	SBR_A_4_FowardDecant_XV26 AT%Q* : BOOL;
	SBR_A_4_ReverseDecant_XV26 AT%Q* : BOOL;
	SBR_A_4_BlowerValve_XV201 AT%Q* : BOOL;
	SBR_A_4_DeSludgeValve_XV241 AT%Q* : BOOL;
	SBR_A_4_SBRValve_XV205 AT%Q* : BOOL;
	SBR_A_4_SBRMixer_XV205 : BOOL;

	SBR_A_4_bEnable_SW : BOOL;
	SBR_A_4_Blower_B201 : BOOL;
	SBR_A_4_DesludgePump_P201 : BOOL;
	SBR_A_4_filling : BOOL;
	SBR_A_4_aeration : BOOL;
	SBR_A_4_settling : BOOL;
	SBR_A_4_decanting : BOOL;
	SBR_A_4_desludging : BOOL;
	SBR_A_4_SBRMixer_M200 : BOOL;
	SBR_A_4_warning_DONotInRange : BOOL;


	SludeTankSensorLevelHi_LSL510A: inBlock;
	SBRReactor_1: SBRReactor;
	SBRReactor_2: SBRReactor;
	SBRReactor_3: SBRReactor;
	SBRReactor_4: SBRReactor;

	SBRMixer_M200A1_A_remote_mode AT%I* : BOOL;
	SBRMixer_M200A1_A_overload AT%I* : BOOL;
	SBRMixer_M200A1_A_incomplete AT%I* : BOOL;
	SBRMixer_M200A1_A_status AT%I* : BOOL;

	SBRMixer_M200A1_A_command AT%Q* : BOOL;

	SBRMixer_M200A1_A_in : BOOL;
	SBRMixer_M200A1_A_overload_error : BOOL;
	SBRMixer_M200A1_A_incomplete_error : BOOL;
	SBRMixer_M200A1_A_status_error : BOOL;
	SBRMixer_M200A1_A_common_error : BOOL;
	SBRMixer_M200A1_A_stop_error : BOOL;

	SBRMixer_M200A1_A_overload_Filter : ErrorFilter;
	SBRMixer_M200A1_A_incomplete_Filter : ErrorFilter;
	SBRMixer_M200A1_A_status_Filter : ErrorFilter;
	SBRMixer_M200A1_A_stop_Filter : ErrorFilter;

	SBRMixer_M200A1_B_remote_mode AT%I* : BOOL;
	SBRMixer_M200A1_B_overload AT%I* : BOOL;
	SBRMixer_M200A1_B_incomplete AT%I* : BOOL;
	SBRMixer_M200A1_B_status AT%I* : BOOL;

	SBRMixer_M200A1_B_command AT%Q* : BOOL;

	SBRMixer_M200A1_B_in : BOOL;
	SBRMixer_M200A1_B_overload_error : BOOL;
	SBRMixer_M200A1_B_incomplete_error : BOOL;
	SBRMixer_M200A1_B_status_error : BOOL;
	SBRMixer_M200A1_B_common_error : BOOL;
	SBRMixer_M200A1_B_stop_error : BOOL;

	SBRMixer_M200A1_B_overload_Filter : ErrorFilter;
	SBRMixer_M200A1_B_incomplete_Filter : ErrorFilter;
	SBRMixer_M200A1_B_status_Filter : ErrorFilter;
	SBRMixer_M200A1_B_stop_Filter : ErrorFilter;


	SBRMixer_M200A1_C_remote_mode AT%I* : BOOL;
	SBRMixer_M200A1_C_overload AT%I* : BOOL;
	SBRMixer_M200A1_C_incomplete AT%I* : BOOL;
	SBRMixer_M200A1_C_status AT%I* : BOOL;

	SBRMixer_M200A1_C_command AT%Q* : BOOL;

	SBRMixer_M200A1_C_in : BOOL;
	SBRMixer_M200A1_C_overload_error : BOOL;
	SBRMixer_M200A1_C_incomplete_error : BOOL;
	SBRMixer_M200A1_C_status_error : BOOL;
	SBRMixer_M200A1_C_common_error : BOOL;
	SBRMixer_M200A1_C_stop_error : BOOL;

	SBRMixer_M200A1_C_overload_Filter : ErrorFilter;
	SBRMixer_M200A1_C_incomplete_Filter : ErrorFilter;
	SBRMixer_M200A1_C_status_Filter : ErrorFilter;
	SBRMixer_M200A1_C_stop_Filter : ErrorFilter;



	SBRMixer_M200A2_A_remote_mode AT%I* : BOOL;
	SBRMixer_M200A2_A_overload AT%I* : BOOL;
	SBRMixer_M200A2_A_incomplete AT%I* : BOOL;
	SBRMixer_M200A2_A_status AT%I* : BOOL;

	SBRMixer_M200A2_A_command AT%Q* : BOOL;

	SBRMixer_M200A2_A_in : BOOL;
	SBRMixer_M200A2_A_overload_error : BOOL;
	SBRMixer_M200A2_A_incomplete_error : BOOL;
	SBRMixer_M200A2_A_status_error : BOOL;
	SBRMixer_M200A2_A_common_error : BOOL;
	SBRMixer_M200A2_A_stop_error : BOOL;

	SBRMixer_M200A2_A_overload_Filter : ErrorFilter;
	SBRMixer_M200A2_A_incomplete_Filter : ErrorFilter;
	SBRMixer_M200A2_A_status_Filter : ErrorFilter;
	SBRMixer_M200A2_A_stop_Filter : ErrorFilter;

	SBRMixer_M200A2_B_remote_mode AT%I* : BOOL;
	SBRMixer_M200A2_B_overload AT%I* : BOOL;
	SBRMixer_M200A2_B_incomplete AT%I* : BOOL;
	SBRMixer_M200A2_B_status AT%I* : BOOL;

	SBRMixer_M200A2_B_command AT%Q* : BOOL;

	SBRMixer_M200A2_B_in : BOOL;
	SBRMixer_M200A2_B_overload_error : BOOL;
	SBRMixer_M200A2_B_incomplete_error : BOOL;
	SBRMixer_M200A2_B_status_error : BOOL;
	SBRMixer_M200A2_B_common_error : BOOL;
	SBRMixer_M200A2_B_stop_error : BOOL;

	SBRMixer_M200A2_B_overload_Filter : ErrorFilter;
	SBRMixer_M200A2_B_incomplete_Filter : ErrorFilter;
	SBRMixer_M200A2_B_status_Filter : ErrorFilter;
	SBRMixer_M200A2_B_stop_Filter : ErrorFilter;


	SBRMixer_M200A2_C_remote_mode AT%I* : BOOL;
	SBRMixer_M200A2_C_overload AT%I* : BOOL;
	SBRMixer_M200A2_C_incomplete AT%I* : BOOL;
	SBRMixer_M200A2_C_status AT%I* : BOOL;

	SBRMixer_M200A2_C_command AT%Q* : BOOL;

	SBRMixer_M200A2_C_in : BOOL;
	SBRMixer_M200A2_C_overload_error : BOOL;
	SBRMixer_M200A2_C_incomplete_error : BOOL;
	SBRMixer_M200A2_C_status_error : BOOL;
	SBRMixer_M200A2_C_common_error : BOOL;
	SBRMixer_M200A2_C_stop_error : BOOL;

	SBRMixer_M200A2_C_overload_Filter : ErrorFilter;
	SBRMixer_M200A2_C_incomplete_Filter : ErrorFilter;
	SBRMixer_M200A2_C_status_Filter : ErrorFilter;
	SBRMixer_M200A2_C_stop_Filter : ErrorFilter;



	SBRMixer_M200A3_A_remote_mode AT%I* : BOOL;
	SBRMixer_M200A3_A_overload AT%I* : BOOL;
	SBRMixer_M200A3_A_incomplete AT%I* : BOOL;
	SBRMixer_M200A3_A_status AT%I* : BOOL;

	SBRMixer_M200A3_A_command AT%Q* : BOOL;

	SBRMixer_M200A3_A_in : BOOL;
	SBRMixer_M200A3_A_overload_error : BOOL;
	SBRMixer_M200A3_A_incomplete_error : BOOL;
	SBRMixer_M200A3_A_status_error : BOOL;
	SBRMixer_M200A3_A_common_error : BOOL;
	SBRMixer_M200A3_A_stop_error : BOOL;

	SBRMixer_M200A3_A_overload_Filter : ErrorFilter;
	SBRMixer_M200A3_A_incomplete_Filter : ErrorFilter;
	SBRMixer_M200A3_A_status_Filter : ErrorFilter;
	SBRMixer_M200A3_A_stop_Filter : ErrorFilter;

	SBRMixer_M200A3_B_remote_mode AT%I* : BOOL;
	SBRMixer_M200A3_B_overload AT%I* : BOOL;
	SBRMixer_M200A3_B_incomplete AT%I* : BOOL;
	SBRMixer_M200A3_B_status AT%I* : BOOL;

	SBRMixer_M200A3_B_command AT%Q* : BOOL;

	SBRMixer_M200A3_B_in : BOOL;
	SBRMixer_M200A3_B_overload_error : BOOL;
	SBRMixer_M200A3_B_incomplete_error : BOOL;
	SBRMixer_M200A3_B_status_error : BOOL;
	SBRMixer_M200A3_B_common_error : BOOL;
	SBRMixer_M200A3_B_stop_error : BOOL;

	SBRMixer_M200A3_B_overload_Filter : ErrorFilter;
	SBRMixer_M200A3_B_incomplete_Filter : ErrorFilter;
	SBRMixer_M200A3_B_status_Filter : ErrorFilter;
	SBRMixer_M200A3_B_stop_Filter : ErrorFilter;


	SBRMixer_M200A3_C_remote_mode AT%I* : BOOL;
	SBRMixer_M200A3_C_overload AT%I* : BOOL;
	SBRMixer_M200A3_C_incomplete AT%I* : BOOL;
	SBRMixer_M200A3_C_status AT%I* : BOOL;

	SBRMixer_M200A3_C_command AT%Q* : BOOL;

	SBRMixer_M200A3_C_in : BOOL;
	SBRMixer_M200A3_C_overload_error : BOOL;
	SBRMixer_M200A3_C_incomplete_error : BOOL;
	SBRMixer_M200A3_C_status_error : BOOL;
	SBRMixer_M200A3_C_common_error : BOOL;
	SBRMixer_M200A3_C_stop_error : BOOL;

	SBRMixer_M200A3_C_overload_Filter : ErrorFilter;
	SBRMixer_M200A3_C_incomplete_Filter : ErrorFilter;
	SBRMixer_M200A3_C_status_Filter : ErrorFilter;
	SBRMixer_M200A3_C_stop_Filter : ErrorFilter;

	DesludgePump_P201A_1_remote_mode AT%I* : BOOL;
	DesludgePump_P201A_1_overload AT%I* : BOOL;
	DesludgePump_P201A_1_incomplete AT%I* : BOOL;
	DesludgePump_P201A_1_status AT%I* : BOOL;

	DesludgePump_P201A_1_command AT%Q* : BOOL;

	DesludgePump_P201A_1_in : BOOL;
	DesludgePump_P201A_1_overload_error : BOOL;
	DesludgePump_P201A_1_incomplete_error : BOOL;
	DesludgePump_P201A_1_status_error : BOOL;
	DesludgePump_P201A_1_common_error : BOOL;
	DesludgePump_P201A_1_stop_error : BOOL;

	DesludgePump_P201A_1_overload_Filter : ErrorFilter;
	DesludgePump_P201A_1_incomplete_Filter : ErrorFilter;
	DesludgePump_P201A_1_status_Filter : ErrorFilter;
	DesludgePump_P201A_1_stop_Filter : ErrorFilter;



	DesludgePump_P201A_2_remote_mode AT%I* : BOOL;
	DesludgePump_P201A_2_overload AT%I* : BOOL;
	DesludgePump_P201A_2_incomplete AT%I* : BOOL;
	DesludgePump_P201A_2_status AT%I* : BOOL;

	DesludgePump_P201A_2_command AT%Q* : BOOL;

	DesludgePump_P201A_2_in : BOOL;
	DesludgePump_P201A_2_overload_error : BOOL;
	DesludgePump_P201A_2_incomplete_error : BOOL;
	DesludgePump_P201A_2_status_error : BOOL;
	DesludgePump_P201A_2_common_error : BOOL;
	DesludgePump_P201A_2_stop_error : BOOL;

	DesludgePump_P201A_2_overload_Filter : ErrorFilter;
	DesludgePump_P201A_2_incomplete_Filter : ErrorFilter;
	DesludgePump_P201A_2_status_Filter : ErrorFilter;
	DesludgePump_P201A_2_stop_Filter : ErrorFilter;

	DesludgePump_P201A :Equipment_Dual;


	Blower_B201A_1_remote_mode AT%I* : BOOL;
	Blower_B201A_1_overload AT%I* : BOOL;
	Blower_B201A_1_incomplete AT%I* : BOOL;
	Blower_B201A_1_status AT%I* : BOOL;

	Blower_B201A_1_command AT%Q* : BOOL;

	Blower_B201A_1_in : BOOL;
	Blower_B201A_1_overload_error : BOOL;
	Blower_B201A_1_incomplete_error : BOOL;
	Blower_B201A_1_status_error : BOOL;
	Blower_B201A_1_common_error : BOOL;
	Blower_B201A_1_stop_error : BOOL;

	Blower_B201A_1_overload_Filter : ErrorFilter;
	Blower_B201A_1_incomplete_Filter : ErrorFilter;
	Blower_B201A_1_status_Filter : ErrorFilter;
	Blower_B201A_1_stop_Filter : ErrorFilter;



	Blower_B201A_2_remote_mode AT%I* : BOOL;
	Blower_B201A_2_overload AT%I* : BOOL;
	Blower_B201A_2_incomplete AT%I* : BOOL;
	Blower_B201A_2_status AT%I* : BOOL;

	Blower_B201A_2_command AT%Q* : BOOL;

	Blower_B201A_2_in : BOOL;
	Blower_B201A_2_overload_error : BOOL;
	Blower_B201A_2_incomplete_error : BOOL;
	Blower_B201A_2_status_error : BOOL;
	Blower_B201A_2_common_error : BOOL;
	Blower_B201A_2_stop_error : BOOL;

	Blower_B201A_2_overload_Filter : ErrorFilter;
	Blower_B201A_2_incomplete_Filter : ErrorFilter;
	Blower_B201A_2_status_Filter : ErrorFilter;
	Blower_B201A_2_stop_Filter : ErrorFilter;



	Blower_B201A_3_remote_mode AT%I* : BOOL;
	Blower_B201A_3_overload AT%I* : BOOL;
	Blower_B201A_3_incomplete AT%I* : BOOL;
	Blower_B201A_3_status AT%I* : BOOL;

	Blower_B201A_3_command AT%Q* : BOOL;

	Blower_B201A_3_in : BOOL;
	Blower_B201A_3_overload_error : BOOL;
	Blower_B201A_3_incomplete_error : BOOL;
	Blower_B201A_3_status_error : BOOL;
	Blower_B201A_3_common_error : BOOL;
	Blower_B201A_3_stop_error : BOOL;

	Blower_B201A_3_overload_Filter : ErrorFilter;
	Blower_B201A_3_incomplete_Filter : ErrorFilter;
	Blower_B201A_3_status_Filter : ErrorFilter;
	Blower_B201A_3_stop_Filter : ErrorFilter;


END_VAR

VAR PERSISTENT
	FILLING_TOKEN : INT;
	AERATION_TOKEN: INT;
	DECANTING_TOKEN: INT;
END_VAR
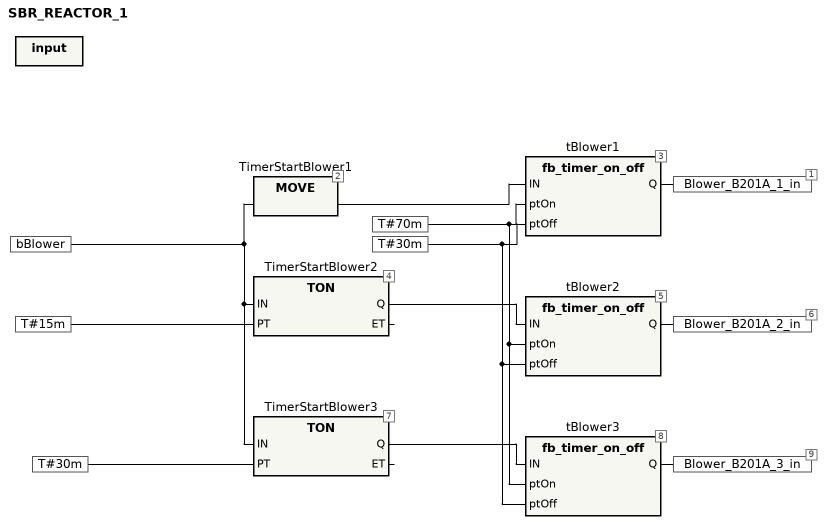
[picture p10: SBR_REACTOR_1 (CFC)]
_CFC_ (* Continuous Function Chart, elements in execution order *)
#0 input()
#1 Blower_B201A_1_in <= #3.Q
#2 TimerStartBlower1:MOVE(bBlower)
#3 tBlower1:fb_timer_on_off(IN: #2, ptOn: T#70m, ptOff: T#30m)
#4 TimerStartBlower2:TON(IN: bBlower, PT: T#15m)
#5 tBlower2:fb_timer_on_off(IN: #4.Q, ptOn: T#70m, ptOff: T#30m)
#6 Blower_B201A_2_in <= #5.Q
#7 TimerStartBlower3:TON(IN: bBlower, PT: T#30m)
#8 tBlower3:fb_timer_on_off(IN: #7.Q, ptOn: T#70m, ptOff: T#30m)
#9 Blower_B201A_3_in <= #8.Q
_END_CFC_
END_PROGRAM
ACTION input:
SludeTankSensorLevelHi_LSL510A();

SBRReactor_1(
	bEnable:=SBR_A_1_bEnable_SW ,
	SludgeTankLevelHi:= SludeTankSensorLevelHi_LSL510A.Q,
	SBRLevelSensor_LSH200:= SBR_A_1_SBRLevelSensor_LSH200,
	rDO201:= SBR_A_1_DOSensor_DO201,
	DecanterLevelSensorHi:=SBR_A_1_DecanterLevelSensorHi_Rx ,
	DecanterLevelSensorLow:=SBR_A_1_DecanterLevelSensorLow_Rx ,
	FILLING_TOKEN:=FILLING_TOKEN ,
	AERATION_TOKEN:= AERATION_TOKEN,
	DECANTING_TOKEN:= DECANTING_TOKEN,
	bBlowerOn=>SBR_A_1_Blower_B201 ,
	bDeSludgePump=>SBR_A_1_DesludgePump_P201 ,
	bFilling=>SBR_A_1_filling ,
	bAeration=>SBR_A_1_aeration ,
	bSettling=>SBR_A_1_settling ,
	bDecanting=>SBR_A_1_decanting ,
	bDesluging=>SBR_A_1_desludging ,
	bWarning_DoNotInRange=>SBR_A_1_warning_DONotInRange ,
	bForwardDecant=>SBR_A_1_FowardDecant_XV26 ,
	bReverseDecant=>SBR_A_1_ReverseDecant_XV26 ,
	bBlowerValve_XV201=>SBR_A_1_BlowerValve_XV201 ,
	bDeslugValve_XV241=> SBR_A_1_DeSludgeValve_XV241,
	bSBRValve_XV205=>SBR_A_1_SBRValve_XV205 ,
	bSBRMixer=>SBR_A_1_SBRMixer_XV205 );


SBRReactor_2(
	bEnable:=SBR_A_2_bEnable_SW ,
	SludgeTankLevelHi:= SludeTankSensorLevelHi_LSL510A.Q,
	SBRLevelSensor_LSH200:= SBR_A_2_SBRLevelSensor_LSH200,
	rDO201:= SBR_A_2_DOSensor_DO201,
	DecanterLevelSensorHi:=SBR_A_2_DecanterLevelSensorHi_Rx ,
	DecanterLevelSensorLow:=SBR_A_2_DecanterLevelSensorLow_Rx ,
	FILLING_TOKEN:=FILLING_TOKEN ,
	AERATION_TOKEN:= AERATION_TOKEN,
	DECANTING_TOKEN:= DECANTING_TOKEN,
	bBlowerOn=>SBR_A_2_Blower_B201 ,
	bDeSludgePump=>SBR_A_2_DesludgePump_P201 ,
	bFilling=>SBR_A_2_filling ,
	bAeration=>SBR_A_2_aeration ,
	bSettling=>SBR_A_2_settling ,
	bDecanting=>SBR_A_2_decanting ,
	bDesluging=>SBR_A_2_desludging ,
	bWarning_DoNotInRange=>SBR_A_2_warning_DONotInRange ,
	bForwardDecant=>SBR_A_2_FowardDecant_XV26 ,
	bReverseDecant=>SBR_A_2_ReverseDecant_XV26 ,
	bBlowerValve_XV201=>SBR_A_2_BlowerValve_XV201 ,
	bDeslugValve_XV241=> SBR_A_2_DeSludgeValve_XV241,
	bSBRValve_XV205=>SBR_A_2_SBRValve_XV205 ,
	bSBRMixer=>SBR_A_2_SBRMixer_XV205 );


SBRReactor_3(
	bEnable:=SBR_A_3_bEnable_SW ,
	SludgeTankLevelHi:= SludeTankSensorLevelHi_LSL510A.Q,
	SBRLevelSensor_LSH200:= SBR_A_3_SBRLevelSensor_LSH200,
	rDO201:= SBR_A_3_DOSensor_DO201,
	DecanterLevelSensorHi:=SBR_A_3_DecanterLevelSensorHi_Rx ,
	DecanterLevelSensorLow:=SBR_A_3_DecanterLevelSensorLow_Rx ,
	FILLING_TOKEN:=FILLING_TOKEN ,
	AERATION_TOKEN:= AERATION_TOKEN,
	DECANTING_TOKEN:= DECANTING_TOKEN,
	bBlowerOn=>SBR_A_3_Blower_B201 ,
	bDeSludgePump=>SBR_A_3_DesludgePump_P201 ,
	bFilling=>SBR_A_3_filling ,
	bAeration=>SBR_A_3_aeration ,
	bSettling=>SBR_A_3_settling ,
	bDecanting=>SBR_A_3_decanting ,
	bDesluging=>SBR_A_3_desludging ,
	bWarning_DoNotInRange=>SBR_A_3_warning_DONotInRange ,
	bForwardDecant=>SBR_A_3_FowardDecant_XV26 ,
	bReverseDecant=>SBR_A_3_ReverseDecant_XV26 ,
	bBlowerValve_XV201=>SBR_A_3_BlowerValve_XV201 ,
	bDeslugValve_XV241=> SBR_A_3_DeSludgeValve_XV241,
	bSBRValve_XV205=>SBR_A_3_SBRValve_XV205 ,
	bSBRMixer=>SBR_A_3_SBRMixer_XV205 );


SBRReactor_4(
	bEnable:=SBR_A_4_bEnable_SW ,
	SludgeTankLevelHi:= SludeTankSensorLevelHi_LSL510A.Q,
	SBRLevelSensor_LSH200:= SBR_A_4_SBRLevelSensor_LSH200,
	rDO201:= SBR_A_4_DOSensor_DO201,
	DecanterLevelSensorHi:=SBR_A_4_DecanterLevelSensorHi_Rx ,
	DecanterLevelSensorLow:=SBR_A_4_DecanterLevelSensorLow_Rx ,
	FILLING_TOKEN:=FILLING_TOKEN ,
	AERATION_TOKEN:= AERATION_TOKEN,
	DECANTING_TOKEN:= DECANTING_TOKEN,
	bBlowerOn=>SBR_A_4_Blower_B201 ,
	bDeSludgePump=>SBR_A_4_DesludgePump_P201 ,
	bFilling=>SBR_A_4_filling ,
	bAeration=>SBR_A_4_aeration ,
	bSettling=>SBR_A_4_settling ,
	bDecanting=>SBR_A_4_decanting ,
	bDesluging=>SBR_A_4_desludging ,
	bWarning_DoNotInRange=>SBR_A_4_warning_DONotInRange ,
	bForwardDecant=>SBR_A_4_FowardDecant_XV26 ,
	bReverseDecant=>SBR_A_4_ReverseDecant_XV26 ,
	bBlowerValve_XV201=>SBR_A_4_BlowerValve_XV201 ,
	bDeslugValve_XV241=> SBR_A_4_DeSludgeValve_XV241,
	bSBRValve_XV205=>SBR_A_4_SBRValve_XV205 ,
	bSBRMixer=>SBR_A_4_SBRMixer_XV205 );


bDeSludge:=SBR_A_1_DeSludgeValve_XV241 OR SBR_A_2_DeSludgeValve_XV241 OR SBR_A_3_DeSludgeValve_XV241 OR SBR_A_4_DeSludgeValve_XV241;
bBlower:= SBR_A_1_Blower_B201 OR SBR_A_2_Blower_B201 OR SBR_A_3_Blower_B201 OR SBR_A_4_Blower_B201;



SBRMixer_M200A1_A_in := SBR_A_1_SBRMixer_XV205;
SBRMixer_M200A1_A_command := SBRMixer_M200A1_A_in AND SBRMixer_M200A1_A_remote_mode;
SBRMixer_M200A1_A_overload_Filter(IN:=(SBRMixer_M200A1_A_overload AND SBRMixer_M200A1_A_in),PT:=T#2s,Q=>SBRMixer_M200A1_A_overload_error);
SBRMixer_M200A1_A_incomplete_Filter(IN:=(SBRMixer_M200A1_A_incomplete AND SBRMixer_M200A1_A_in),PT:=T#2s,Q=>SBRMixer_M200A1_A_incomplete_error);
SBRMixer_M200A1_A_status_Filter(IN:=(NOT SBRMixer_M200A1_A_status AND SBRMixer_M200A1_A_in),PT:=T#10s, Q=>SBRMixer_M200A1_A_status_error);
SBRMixer_M200A1_A_stop_Filter(IN:=( SBRMixer_M200A1_A_status AND NOT SBRMixer_M200A1_A_in),PT:=T#10s, Q=>SBRMixer_M200A1_A_stop_error);

SBRMixer_M200A1_A_common_error := SBRMixer_M200A1_A_overload_error OR SBRMixer_M200A1_A_incomplete_error OR SBRMixer_M200A1_A_status_error OR SBRMixer_M200A1_A_stop_error;


SBRMixer_M200A1_B_in := SBR_A_1_SBRMixer_XV205;
SBRMixer_M200A1_B_command := SBRMixer_M200A1_B_in AND SBRMixer_M200A1_B_remote_mode;
SBRMixer_M200A1_B_overload_Filter(IN:=(SBRMixer_M200A1_B_overload AND SBRMixer_M200A1_B_in),PT:=T#2s,Q=>SBRMixer_M200A1_B_overload_error);
SBRMixer_M200A1_B_incomplete_Filter(IN:=(SBRMixer_M200A1_B_incomplete AND SBRMixer_M200A1_B_in),PT:=T#2s,Q=>SBRMixer_M200A1_B_incomplete_error);
SBRMixer_M200A1_B_status_Filter(IN:=(NOT SBRMixer_M200A1_B_status AND SBRMixer_M200A1_B_in),PT:=T#10s, Q=>SBRMixer_M200A1_B_status_error);
SBRMixer_M200A1_B_stop_Filter(IN:=( SBRMixer_M200A1_B_status AND NOT SBRMixer_M200A1_B_in),PT:=T#10s, Q=>SBRMixer_M200A1_B_stop_error);

SBRMixer_M200A1_B_common_error := SBRMixer_M200A1_B_overload_error OR SBRMixer_M200A1_B_incomplete_error OR SBRMixer_M200A1_B_status_error OR SBRMixer_M200A1_B_stop_error;


SBRMixer_M200A1_C_in := SBR_A_1_SBRMixer_XV205;
SBRMixer_M200A1_C_command := SBRMixer_M200A1_C_in AND SBRMixer_M200A1_C_remote_mode;
SBRMixer_M200A1_C_overload_Filter(IN:=(SBRMixer_M200A1_C_overload AND SBRMixer_M200A1_C_in),PT:=T#2s,Q=>SBRMixer_M200A1_C_overload_error);
SBRMixer_M200A1_C_incomplete_Filter(IN:=(SBRMixer_M200A1_C_incomplete AND SBRMixer_M200A1_C_in),PT:=T#2s,Q=>SBRMixer_M200A1_C_incomplete_error);
SBRMixer_M200A1_C_status_Filter(IN:=(NOT SBRMixer_M200A1_C_status AND SBRMixer_M200A1_C_in),PT:=T#10s, Q=>SBRMixer_M200A1_C_status_error);
SBRMixer_M200A1_C_stop_Filter(IN:=( SBRMixer_M200A1_C_status AND NOT SBRMixer_M200A1_C_in),PT:=T#10s, Q=>SBRMixer_M200A1_C_stop_error);

SBRMixer_M200A1_C_common_error := SBRMixer_M200A1_C_overload_error OR SBRMixer_M200A1_C_incomplete_error OR SBRMixer_M200A1_C_status_error OR SBRMixer_M200A1_C_stop_error;



SBRMixer_M200A2_A_in := SBR_A_2_SBRMixer_XV205;
SBRMixer_M200A2_A_command := SBRMixer_M200A2_A_in AND SBRMixer_M200A2_A_remote_mode;
SBRMixer_M200A2_A_overload_Filter(IN:=(SBRMixer_M200A2_A_overload AND SBRMixer_M200A2_A_in),PT:=T#2s,Q=>SBRMixer_M200A2_A_overload_error);
SBRMixer_M200A2_A_incomplete_Filter(IN:=(SBRMixer_M200A2_A_incomplete AND SBRMixer_M200A2_A_in),PT:=T#2s,Q=>SBRMixer_M200A2_A_incomplete_error);
SBRMixer_M200A2_A_status_Filter(IN:=(NOT SBRMixer_M200A2_A_status AND SBRMixer_M200A2_A_in),PT:=T#10s, Q=>SBRMixer_M200A2_A_status_error);
SBRMixer_M200A2_A_stop_Filter(IN:=( SBRMixer_M200A2_A_status AND NOT SBRMixer_M200A2_A_in),PT:=T#10s, Q=>SBRMixer_M200A2_A_stop_error);

SBRMixer_M200A2_A_common_error := SBRMixer_M200A2_A_overload_error OR SBRMixer_M200A2_A_incomplete_error OR SBRMixer_M200A2_A_status_error OR SBRMixer_M200A2_A_stop_error;


SBRMixer_M200A2_B_in := SBR_A_2_SBRMixer_XV205;
SBRMixer_M200A2_B_command := SBRMixer_M200A2_B_in AND SBRMixer_M200A2_B_remote_mode;
SBRMixer_M200A2_B_overload_Filter(IN:=(SBRMixer_M200A2_B_overload AND SBRMixer_M200A2_B_in),PT:=T#2s,Q=>SBRMixer_M200A2_B_overload_error);
SBRMixer_M200A2_B_incomplete_Filter(IN:=(SBRMixer_M200A2_B_incomplete AND SBRMixer_M200A2_B_in),PT:=T#2s,Q=>SBRMixer_M200A2_B_incomplete_error);
SBRMixer_M200A2_B_status_Filter(IN:=(NOT SBRMixer_M200A2_B_status AND SBRMixer_M200A2_B_in),PT:=T#10s, Q=>SBRMixer_M200A2_B_status_error);
SBRMixer_M200A1_B_stop_Filter(IN:=( SBRMixer_M200A1_B_status AND NOT SBRMixer_M200A1_B_in),PT:=T#10s, Q=>SBRMixer_M200A1_B_stop_error);

SBRMixer_M200A1_B_common_error := SBRMixer_M200A1_B_overload_error OR SBRMixer_M200A1_B_incomplete_error OR SBRMixer_M200A1_B_status_error OR SBRMixer_M200A1_B_stop_error;


SBRMixer_M200A2_C_in := SBR_A_2_SBRMixer_XV205;
SBRMixer_M200A2_C_command := SBRMixer_M200A2_C_in AND SBRMixer_M200A2_C_remote_mode;
SBRMixer_M200A2_C_overload_Filter(IN:=(SBRMixer_M200A2_C_overload AND SBRMixer_M200A2_C_in),PT:=T#2s,Q=>SBRMixer_M200A2_C_overload_error);
SBRMixer_M200A2_C_incomplete_Filter(IN:=(SBRMixer_M200A2_C_incomplete AND SBRMixer_M200A2_C_in),PT:=T#2s,Q=>SBRMixer_M200A2_C_incomplete_error);
SBRMixer_M200A2_C_status_Filter(IN:=(NOT SBRMixer_M200A2_C_status AND SBRMixer_M200A2_C_in),PT:=T#10s, Q=>SBRMixer_M200A2_C_status_error);
SBRMixer_M200A2_C_stop_Filter(IN:=( SBRMixer_M200A2_C_status AND NOT SBRMixer_M200A2_C_in),PT:=T#10s, Q=>SBRMixer_M200A2_C_stop_error);

SBRMixer_M200A2_C_common_error := SBRMixer_M200A2_C_overload_error OR SBRMixer_M200A2_C_incomplete_error OR SBRMixer_M200A2_C_status_error OR SBRMixer_M200A2_C_stop_error;



SBRMixer_M200A3_A_in := SBR_A_3_SBRMixer_XV205;
SBRMixer_M200A3_A_command := SBRMixer_M200A3_A_in AND SBRMixer_M200A3_A_remote_mode;
SBRMixer_M200A3_A_overload_Filter(IN:=(SBRMixer_M200A3_A_overload AND SBRMixer_M200A3_A_in),PT:=T#2s,Q=>SBRMixer_M200A3_A_overload_error);
SBRMixer_M200A3_A_incomplete_Filter(IN:=(SBRMixer_M200A3_A_incomplete AND SBRMixer_M200A3_A_in),PT:=T#2s,Q=>SBRMixer_M200A3_A_incomplete_error);
SBRMixer_M200A3_A_status_Filter(IN:=(NOT SBRMixer_M200A3_A_status AND SBRMixer_M200A3_A_in),PT:=T#10s, Q=>SBRMixer_M200A3_A_status_error);
SBRMixer_M200A3_A_stop_Filter(IN:=( SBRMixer_M200A3_A_status AND NOT SBRMixer_M200A3_A_in),PT:=T#10s, Q=>SBRMixer_M200A3_A_stop_error);

SBRMixer_M200A3_A_common_error := SBRMixer_M200A3_A_overload_error OR SBRMixer_M200A3_A_incomplete_error OR SBRMixer_M200A3_A_status_error OR SBRMixer_M200A3_A_stop_error;


SBRMixer_M200A3_B_in := SBR_A_3_SBRMixer_XV205;
SBRMixer_M200A3_B_command := SBRMixer_M200A3_B_in AND SBRMixer_M200A3_B_remote_mode;
SBRMixer_M200A3_B_overload_Filter(IN:=(SBRMixer_M200A3_B_overload AND SBRMixer_M200A3_B_in),PT:=T#2s,Q=>SBRMixer_M200A3_B_overload_error);
SBRMixer_M200A3_B_incomplete_Filter(IN:=(SBRMixer_M200A3_B_incomplete AND SBRMixer_M200A3_B_in),PT:=T#2s,Q=>SBRMixer_M200A3_B_incomplete_error);
SBRMixer_M200A3_B_status_Filter(IN:=(NOT SBRMixer_M200A3_B_status AND SBRMixer_M200A3_B_in),PT:=T#10s, Q=>SBRMixer_M200A3_B_status_error);
SBRMixer_M200A1_B_stop_Filter(IN:=( SBRMixer_M200A1_B_status AND NOT SBRMixer_M200A1_B_in),PT:=T#10s, Q=>SBRMixer_M200A1_B_stop_error);

SBRMixer_M200A1_B_common_error := SBRMixer_M200A1_B_overload_error OR SBRMixer_M200A1_B_incomplete_error OR SBRMixer_M200A1_B_status_error OR SBRMixer_M200A1_B_stop_error;


SBRMixer_M200A3_C_in := SBR_A_3_SBRMixer_XV205;
SBRMixer_M200A3_C_command := SBRMixer_M200A3_C_in AND SBRMixer_M200A3_C_remote_mode;
SBRMixer_M200A3_C_overload_Filter(IN:=(SBRMixer_M200A3_C_overload AND SBRMixer_M200A3_C_in),PT:=T#2s,Q=>SBRMixer_M200A3_C_overload_error);
SBRMixer_M200A3_C_incomplete_Filter(IN:=(SBRMixer_M200A3_C_incomplete AND SBRMixer_M200A3_C_in),PT:=T#2s,Q=>SBRMixer_M200A3_C_incomplete_error);
SBRMixer_M200A3_C_status_Filter(IN:=(NOT SBRMixer_M200A3_C_status AND SBRMixer_M200A3_C_in),PT:=T#10s, Q=>SBRMixer_M200A3_C_status_error);
SBRMixer_M200A3_C_stop_Filter(IN:=( SBRMixer_M200A3_C_status AND NOT SBRMixer_M200A3_C_in),PT:=T#10s, Q=>SBRMixer_M200A3_C_stop_error);

SBRMixer_M200A3_C_common_error := SBRMixer_M200A3_C_overload_error OR SBRMixer_M200A3_C_incomplete_error OR SBRMixer_M200A3_C_status_error OR SBRMixer_M200A3_C_stop_error;



DesludgePump_P201A_1_overload_Filter(IN:=(DesludgePump_P201A_1_overload AND DesludgePump_P201A_1_in),PT:=T#2s,Q=>DesludgePump_P201A_1_overload_error);
DesludgePump_P201A_1_incomplete_Filter(IN:=(DesludgePump_P201A_1_incomplete AND DesludgePump_P201A_1_in),PT:=T#2s,Q=>DesludgePump_P201A_1_incomplete_error);
DesludgePump_P201A_1_status_Filter(IN:=(NOT DesludgePump_P201A_1_status AND DesludgePump_P201A_1_in),PT:=T#10s, Q=>DesludgePump_P201A_1_status_error);
DesludgePump_P201A_1_stop_Filter(IN:=( DesludgePump_P201A_1_status AND NOT DesludgePump_P201A_1_in),PT:=T#10s, Q=>DesludgePump_P201A_1_stop_error);

DesludgePump_P201A_1_common_error := DesludgePump_P201A_1_overload_error OR DesludgePump_P201A_1_incomplete_error OR DesludgePump_P201A_1_status_error OR DesludgePump_P201A_1_stop_error;


DesludgePump_P201A_2_overload_Filter(IN:=(DesludgePump_P201A_2_overload AND DesludgePump_P201A_2_in),PT:=T#2s,Q=>DesludgePump_P201A_2_overload_error);
DesludgePump_P201A_2_incomplete_Filter(IN:=(DesludgePump_P201A_2_incomplete AND DesludgePump_P201A_2_in),PT:=T#2s,Q=>DesludgePump_P201A_2_incomplete_error);
DesludgePump_P201A_2_status_Filter(IN:=(NOT DesludgePump_P201A_2_status AND DesludgePump_P201A_2_in),PT:=T#10s, Q=>DesludgePump_P201A_2_status_error);
DesludgePump_P201A_2_stop_Filter(IN:=( DesludgePump_P201A_2_status AND NOT DesludgePump_P201A_2_in),PT:=T#10s, Q=>DesludgePump_P201A_2_stop_error);

DesludgePump_P201A_2_common_error := DesludgePump_P201A_2_overload_error OR DesludgePump_P201A_2_incomplete_error OR DesludgePump_P201A_2_status_error OR DesludgePump_P201A_2_stop_error;

DesludgePump_P201A_1_in := bDeSludge;
DesludgePump_P201A(
	ERROR1:=DesludgePump_P201A_1_common_error ,
	ERROR2:=DesludgePump_P201A_2_common_error ,
	remote1:=DesludgePump_P201A_1_remote_mode ,
	remote2:=DesludgePump_P201A_2_remote_mode ,
	IN1:=DesludgePump_P201A_1_in ,
	IN2:=DesludgePump_P201A_2_in ,
	Command1=>DesludgePump_P201A_1_command,
	Command2=>DesludgePump_P201A_2_command );


Blower_B201A_1_command := Blower_B201A_1_in AND Blower_B201A_1_remote_mode;
Blower_B201A_1_overload_Filter(IN:=(Blower_B201A_1_overload AND Blower_B201A_1_in),PT:=T#2s,Q=>Blower_B201A_1_overload_error);
Blower_B201A_1_incomplete_Filter(IN:=(Blower_B201A_1_incomplete AND Blower_B201A_1_in),PT:=T#2s,Q=>Blower_B201A_1_incomplete_error);
Blower_B201A_1_status_Filter(IN:=(NOT Blower_B201A_1_status AND Blower_B201A_1_in),PT:=T#10s, Q=>Blower_B201A_1_status_error);
Blower_B201A_1_stop_Filter(IN:=( Blower_B201A_1_status AND NOT Blower_B201A_1_in),PT:=T#10s, Q=>Blower_B201A_1_stop_error);

Blower_B201A_1_common_error := Blower_B201A_1_overload_error OR Blower_B201A_1_incomplete_error OR Blower_B201A_1_status_error OR Blower_B201A_1_stop_error;


Blower_B201A_2_command := Blower_B201A_2_in AND Blower_B201A_2_remote_mode;
Blower_B201A_2_overload_Filter(IN:=(Blower_B201A_2_overload AND Blower_B201A_2_in),PT:=T#2s,Q=>Blower_B201A_2_overload_error);
Blower_B201A_2_incomplete_Filter(IN:=(Blower_B201A_2_incomplete AND Blower_B201A_2_in),PT:=T#2s,Q=>Blower_B201A_2_incomplete_error);
Blower_B201A_2_status_Filter(IN:=(NOT Blower_B201A_2_status AND Blower_B201A_2_in),PT:=T#10s, Q=>Blower_B201A_2_status_error);
Blower_B201A_2_stop_Filter(IN:=( Blower_B201A_2_status AND NOT Blower_B201A_2_in),PT:=T#10s, Q=>Blower_B201A_2_stop_error);

Blower_B201A_2_common_error := Blower_B201A_2_overload_error OR Blower_B201A_2_incomplete_error OR Blower_B201A_2_status_error OR Blower_B201A_2_stop_error;


Blower_B201A_3_command := Blower_B201A_3_in AND Blower_B201A_3_remote_mode;
Blower_B201A_3_overload_Filter(IN:=(Blower_B201A_3_overload AND Blower_B201A_3_in),PT:=T#2s,Q=>Blower_B201A_3_overload_error);
Blower_B201A_3_incomplete_Filter(IN:=(Blower_B201A_3_incomplete AND Blower_B201A_3_in),PT:=T#2s,Q=>Blower_B201A_3_incomplete_error);
Blower_B201A_3_status_Filter(IN:=(NOT Blower_B201A_3_status AND Blower_B201A_3_in),PT:=T#10s, Q=>Blower_B201A_3_status_error);
Blower_B201A_3_stop_Filter(IN:=( Blower_B201A_3_status AND NOT Blower_B201A_3_in),PT:=T#10s, Q=>Blower_B201A_3_stop_error);

Blower_B201A_3_common_error := Blower_B201A_3_overload_error OR Blower_B201A_3_incomplete_error OR Blower_B201A_3_status_error OR Blower_B201A_3_stop_error;
END_ACTION

(* POU STREAM_INLET_MIXER_2, CFC *)
PROGRAM STREAM_INLET_MIXER_2
VAR
	LSL101B : inBlock;
	LSS101B : inBlock;
	LSH101B : inBlock;
	LSD101B : inBlock;
	LSL100B : inBlock;
	LSHL100B:inBlock;

	bCriticalEQFloatHi: BOOL;
	bWarningFloatSensorLow: BOOL;
	bCriticalFloatSensorDry: BOOL;



	EQPump_P101B_1_remote_mode AT%I* : BOOL;
	EQPump_P101B_1_overload AT%I* : BOOL;
	EQPump_P101B_1_incomplete AT%I* : BOOL;
	EQPump_P101B_1_status AT%I* : BOOL;

	EQPump_P101B_1_command AT%Q* : BOOL;

	EQPump_P101B_1_in : BOOL;
	EQPump_P101B_1_overload_error : BOOL;
	EQPump_P101B_1_incomplete_error : BOOL;
	EQPump_P101B_1_status_error : BOOL;
	EQPump_P101B_1_common_error : BOOL;
	EQPump_P101B_1_stop_error : BOOL;

	EQPump_P101B_1_overload_Filter : ErrorFilter;
	EQPump_P101B_1_incomplete_Filter : ErrorFilter;
	EQPump_P101B_1_status_Filter : ErrorFilter;
	EQPump_P101B_1_stop_Filter : ErrorFilter;



	EQPump_P101B_2_remote_mode AT%I* : BOOL;
	EQPump_P101B_2_overload AT%I* : BOOL;
	EQPump_P101B_2_incomplete AT%I* : BOOL;
	EQPump_P101B_2_status AT%I* : BOOL;

	EQPump_P101B_2_command AT%Q* : BOOL;

	EQPump_P101B_2_in : BOOL;
	EQPump_P101B_2_overload_error : BOOL;
	EQPump_P101B_2_incomplete_error : BOOL;
	EQPump_P101B_2_status_error : BOOL;
	EQPump_P101B_2_common_error : BOOL;
	EQPump_P101B_2_stop_error : BOOL;

	EQPump_P101B_2_overload_Filter : ErrorFilter;
	EQPump_P101B_2_incomplete_Filter : ErrorFilter;
	EQPump_P101B_2_status_Filter : ErrorFilter;
	EQPump_P101B_2_stop_Filter : ErrorFilter;

	EQPump_P101B_CriticalStartError : BOOL;

	Mixer_M101B_1_remote_mode AT%I* : BOOL;
	Mixer_M101B_1_overload AT%I* : BOOL;
	Mixer_M101B_1_incomplete AT%I* : BOOL;
	Mixer_M101B_1_status AT%I* : BOOL;

	Mixer_M101B_1_command AT%Q* : BOOL;

	Mixer_M101B_1_in : BOOL;
	Mixer_M101B_1_overload_error : BOOL;
	Mixer_M101B_1_incomplete_error : BOOL;
	Mixer_M101B_1_status_error : BOOL;
	Mixer_M101B_1_common_error : BOOL;
	Mixer_M101B_1_stop_error : BOOL;


	Mixer_M101B_1_overload_Filter : ErrorFilter;
	Mixer_M101B_1_incomplete_Filter : ErrorFilter;
	Mixer_M101B_1_status_Filter : ErrorFilter;
	Mixer_M101B_1_stop_Filter : ErrorFilter;


	Mixer_M101B_2_remote_mode AT%I* : BOOL;
	Mixer_M101B_2_overload AT%I* : BOOL;
	Mixer_M101B_2_incomplete AT%I* : BOOL;
	Mixer_M101B_2_status AT%I* : BOOL;

	Mixer_M101B_2_command AT%Q* : BOOL;

	Mixer_M101B_2_in : BOOL;
	Mixer_M101B_2_overload_error : BOOL;
	Mixer_M101B_2_incomplete_error : BOOL;
	Mixer_M101B_2_status_error : BOOL;
	Mixer_M101B_2_common_error : BOOL;
	Mixer_M101B_2_stop_error : BOOL;

	Mixer_M101B_2_overload_Filter : ErrorFilter;
	Mixer_M101B_2_incomplete_Filter : ErrorFilter;
	Mixer_M101B_2_status_Filter : ErrorFilter;
	Mixer_M101B_2_stop_Filter : ErrorFilter;

	Mixer_M101B_CriticalStartEror : BOOL;

	InletPump :Equipment_Dual;
	Mixer :Equipment_Dual;



END_VAR
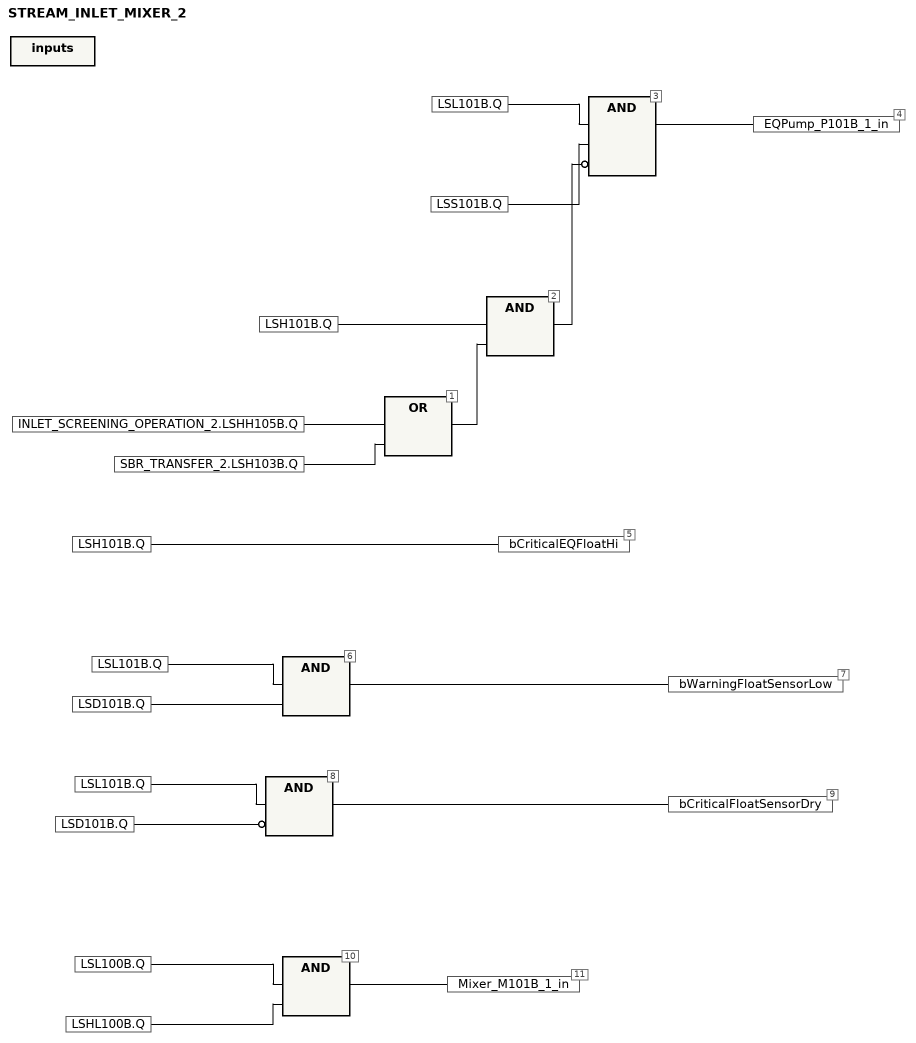
_CFC_ (* Continuous Function Chart, elements in execution order *)
#0 inputs()
#1 OR(INLET_SCREENING_OPERATION_2.LSHH105B.Q, SBR_TRANSFER_2.LSH103B.Q)
#2 AND(LSH101B.Q, #1)
#3 AND(LSL101B.Q, LSS101B.Q, NOT #2)
#4 EQPump_P101B_1_in <= #3
#5 bCriticalEQFloatHi <= LSH101B.Q
#6 AND(LSL101B.Q, LSD101B.Q)
#7 bWarningFloatSensorLow <= #6
#8 AND(LSL101B.Q, NOT LSD101B.Q)
#9 bCriticalFloatSensorDry <= #8
#10 AND(LSL100B.Q, LSHL100B.Q)
#11 Mixer_M101B_1_in <= #10
_END_CFC_
(* the same logic as Structured Text *)
inputs();
EQPump_P101B_1_in := LSL101B.Q AND LSS101B.Q AND NOT (LSH101B.Q AND (INLET_SCREENING_OPERATION_2.LSHH105B.Q OR SBR_TRANSFER_2.LSH103B.Q));
bCriticalEQFloatHi := LSH101B.Q;
bWarningFloatSensorLow := LSL101B.Q AND LSD101B.Q;
bCriticalFloatSensorDry := LSL101B.Q AND NOT LSD101B.Q;
Mixer_M101B_1_in := LSL100B.Q AND LSHL100B.Q;
END_PROGRAM
ACTION inputs:
	LSL101B();
	LSS101B();
	LSH101B();
	LSD101B();

	LSL100B();
	LSHL100B();



EQPump_P101B_1_overload_Filter(IN:=(EQPump_P101B_1_overload AND EQPump_P101B_1_in),PT:=T#10s,Q=>EQPump_P101B_1_overload_error);
EQPump_P101B_1_incomplete_Filter(IN:=(EQPump_P101B_1_incomplete AND EQPump_P101B_1_in),PT:=T#2s,Q=>EQPump_P101B_1_incomplete_error);
EQPump_P101B_1_status_Filter(IN:=(NOT EQPump_P101B_1_status AND EQPump_P101B_1_in),PT:=T#2s, Q=>EQPump_P101B_1_status_error);
EQPump_P101B_1_stop_Filter(IN:=( EQPump_P101B_1_status AND NOT EQPump_P101B_1_in),PT:=T#10s, Q=>EQPump_P101B_1_stop_error);

EQPump_P101B_1_common_error := EQPump_P101B_1_overload_error OR EQPump_P101B_1_incomplete_error OR EQPump_P101B_1_status_error OR EQPump_P101B_1_stop_error;



EQPump_P101B_2_overload_Filter(IN:=(EQPump_P101B_2_overload AND EQPump_P101B_2_in),PT:=T#10s,Q=>EQPump_P101B_2_overload_error);
EQPump_P101B_2_incomplete_Filter(IN:=(EQPump_P101B_2_incomplete AND EQPump_P101B_2_in),PT:=T#2s,Q=>EQPump_P101B_2_incomplete_error);
EQPump_P101B_2_status_Filter(IN:=(NOT EQPump_P101B_2_status AND EQPump_P101B_2_in),PT:=T#2s, Q=>EQPump_P101B_2_status_error);
EQPump_P101B_2_stop_Filter(IN:=( EQPump_P101B_2_status AND NOT EQPump_P101B_2_in),PT:=T#10s, Q=>EQPump_P101B_2_stop_error);

EQPump_P101B_2_common_error := EQPump_P101B_2_overload_error OR EQPump_P101B_2_incomplete_error OR EQPump_P101B_2_status_error OR EQPump_P101B_2_stop_error;

InletPump(
	ERROR1:=EQPump_P101B_1_common_error ,
	ERROR2:=EQPump_P101B_2_common_error ,
	remote1:=EQPump_P101B_1_remote_mode ,
	remote2:= EQPump_P101B_2_remote_mode,
	IN1:=EQPump_P101B_1_in ,
	IN2:=EQPump_P101B_2_in ,
	Command1=>EQPump_P101B_1_command ,
	Command2=>EQPump_P101B_2_command );

EQPump_P101B_CriticalStartError := EQPump_P101B_1_common_error AND EQPump_P101B_2_common_error;


Mixer_M101B_1_overload_Filter(IN:=(Mixer_M101B_1_overload AND Mixer_M101B_1_in),PT:=T#10s,Q=>Mixer_M101B_1_overload_error);
Mixer_M101B_1_incomplete_Filter(IN:=(Mixer_M101B_1_incomplete AND Mixer_M101B_1_in),PT:=T#2s,Q=>Mixer_M101B_1_incomplete_error);
Mixer_M101B_1_status_Filter(IN:=(NOT Mixer_M101B_1_status AND Mixer_M101B_1_in),PT:=T#2s, Q=>Mixer_M101B_1_status_error);
Mixer_M101B_1_stop_Filter(IN:=( Mixer_M101B_1_status AND NOT Mixer_M101B_1_in),PT:=T#10s, Q=>Mixer_M101B_1_stop_error);

Mixer_M101B_1_common_error := Mixer_M101B_1_overload_error OR Mixer_M101B_1_incomplete_error OR Mixer_M101B_1_status_error OR Mixer_M101B_1_stop_error;


Mixer_M101B_2_overload_Filter(IN:=(Mixer_M101B_2_overload AND Mixer_M101B_2_in),PT:=T#10s,Q=>Mixer_M101B_2_overload_error);
Mixer_M101B_2_incomplete_Filter(IN:=(Mixer_M101B_2_incomplete AND Mixer_M101B_2_in),PT:=T#2s,Q=>Mixer_M101B_2_incomplete_error);
Mixer_M101B_2_status_Filter(IN:=(NOT Mixer_M101B_2_status AND Mixer_M101B_2_in),PT:=T#2s, Q=>Mixer_M101B_2_status_error);
Mixer_M101B_2_stop_Filter(IN:=( Mixer_M101B_2_status AND NOT Mixer_M101B_2_in),PT:=T#10s, Q=>Mixer_M101B_2_stop_error);

Mixer_M101B_2_common_error := Mixer_M101B_2_overload_error OR Mixer_M101B_2_incomplete_error OR Mixer_M101B_2_status_error OR Mixer_M101B_2_stop_error;

Mixer(
	ERROR1:=Mixer_M101B_1_common_error ,
	ERROR2:=Mixer_M101B_2_common_error ,
	remote1:=Mixer_M101B_1_remote_mode ,
	remote2:= Mixer_M101B_2_remote_mode,
	IN1:=Mixer_M101B_1_in ,
	IN2:=Mixer_M101B_2_in ,
	Command1=>Mixer_M101B_1_command,
	Command2=>Mixer_M101B_2_command );

Mixer_M101B_CriticalStartEror := Mixer_M101B_1_common_error AND Mixer_M101B_2_common_error;
END_ACTION

(* POU INLET_SCREENING_OPERATION_2, CFC *)
PROGRAM INLET_SCREENING_OPERATION_2
VAR

	LSH105B : inBlock;
	LSHH105B: inBlock;
	Timer1: TON;
	StopTimer: TON;
	timerCompactor: TON;
	bFineScreenDual: BOOL;

	bWarningStreamLineOverflow: BOOL;


	Penstock_PS101B_1_status AT%I* : BOOL;
	Penstock_PS101B_1_command AT%Q* : BOOL;

	Penstock_PS101B_1_in : BOOL;
	Penstock_PS101B_1_open_error : BOOL;
	Penstock_PS101B_1_common_error : BOOL;
	Penstock_PS101B_1_close_error : BOOL;

	Penstock_PS101B_1_open_Filter : ErrorFilter;
	Penstock_PS101B_1_close_Filter : ErrorFilter;




	Penstock_PS101B_2_status AT%I* : BOOL;

	Penstock_PS101B_2_command AT%Q* : BOOL;

	Penstock_PS101B_2_in : BOOL;
	Penstock_PS101B_2_open_error : BOOL;
	Penstock_PS101B_2_common_error : BOOL;
	Penstock_PS101B_2_close_error : BOOL;

	Penstock_PS101B_2_open_Filter : ErrorFilter;
	Penstock_PS101B_2_close_Filter : ErrorFilter;


	Finescreen_F101B_1_remote_mode AT%I* : BOOL;
	Finescreen_F101B_1_overload AT%I* : BOOL;
	Finescreen_F101B_1_incomplete AT%I* : BOOL;
	Finescreen_F101B_1_status AT%I* : BOOL;

	Finescreen_F101B_1_command AT%Q* : BOOL;

	Finescreen_F101B_1_in : BOOL;
	Finescreen_F101B_1_overload_error : BOOL;
	Finescreen_F101B_1_incomplete_error : BOOL;
	Finescreen_F101B_1_status_error : BOOL;
	Finescreen_F101B_1_common_error : BOOL;
	Finescreen_F101B_1_stop_error : BOOL;

	Finescreen_F101B_1_overload_Filter : ErrorFilter;
	Finescreen_F101B_1_incomplete_Filter : ErrorFilter;
	Finescreen_F101B_1_status_Filter : ErrorFilter;
	Finescreen_F101B_1_stop_Filter : ErrorFilter;



	Finescreen_F101B_2_remote_mode AT%I* : BOOL;
	Finescreen_F101B_2_overload AT%I* : BOOL;
	Finescreen_F101B_2_incomplete AT%I* : BOOL;
	Finescreen_F101B_2_status AT%I* : BOOL;

	Finescreen_F101B_2_command AT%Q* : BOOL;

	Finescreen_F101B_2_in : BOOL;
	Finescreen_F101B_2_overload_error : BOOL;
	Finescreen_F101B_2_incomplete_error : BOOL;
	Finescreen_F101B_2_status_error : BOOL;
	Finescreen_F101B_2_common_error : BOOL;
	Finescreen_F101B_2_stop_error : BOOL;

	Finescreen_F101B_2_overload_Filter : ErrorFilter;
	Finescreen_F101B_2_incomplete_Filter : ErrorFilter;
	Finescreen_F101B_2_status_Filter : ErrorFilter;
	Finescreen_F101B_2_stop_Filter : ErrorFilter;

	FineScreen :Equipment_Dual;


	WaterSprayScreen_XV101B_1_open_status AT%I* : BOOL;
	WaterSprayScreen_XV101B_1_close_status AT%I* : BOOL;

	WaterSprayScreen_XV101B_1_command AT%Q* : BOOL;

	WaterSprayScreen_XV101B_1_in : BOOL;
	WaterSprayScreen_XV101B_1_open_error : BOOL;
	WaterSprayScreen_XV101B_1_common_error : BOOL;
	WaterSprayScreen_XV101B_1_close_error : BOOL;

	WaterSprayScreen_XV101B_1_open_Filter : ErrorFilter;
	WaterSprayScreen_XV101B_1_close_Filter : ErrorFilter;



	WaterSprayScreen_XV101B_2_open_status AT%I* : BOOL;
	WaterSprayScreen_XV101B_2_close_status AT%I* : BOOL;

	WaterSprayScreen_XV101B_2_command AT%Q* : BOOL;

	WaterSprayScreen_XV101B_2_in : BOOL;
	WaterSprayScreen_XV101B_2_open_error : BOOL;
	WaterSprayScreen_XV101B_2_common_error : BOOL;
	WaterSprayScreen_XV101B_2_close_error : BOOL;

	WaterSprayScreen_XV101B_2_open_Filter : ErrorFilter;
	WaterSprayScreen_XV101B_2_close_Filter : ErrorFilter;




	WaterSprayScreen1: Equipment_Timed;
	WaterSprayScreen2: Equipment_Timed;



	ScrewConveyer_C102A_remote_mode AT%I* : BOOL;
	ScrewConveyer_C102A_overload AT%I* : BOOL;
	ScrewConveyer_C102A_incomplete AT%I* : BOOL;
	ScrewConveyer_C102A_status AT%I* : BOOL;

	ScrewConveyer_C102A_command AT%Q* : BOOL;

	ScrewConveyer_C102A_in : BOOL;
	ScrewConveyer_C102A_overload_error : BOOL;
	ScrewConveyer_C102A_incomplete_error : BOOL;
	ScrewConveyer_C102A_status_error : BOOL;
	ScrewConveyer_C102A_common_error : BOOL;
	ScrewConveyer_C102A_stop_error : BOOL;

	ScrewConveyer_C102A_overload_Filter : ErrorFilter;
	ScrewConveyer_C102A_incomplete_Filter : ErrorFilter;
	ScrewConveyer_C102A_status_Filter : ErrorFilter;
	ScrewConveyer_C102A_stop_Filter : ErrorFilter;

	ScreenCompactor_C101B_remote_mode AT%I* : BOOL;
	ScreenCompactor_C101B_overload AT%I* : BOOL;
	ScreenCompactor_C101B_incomplete AT%I* : BOOL;
	ScreenCompactor_C101B_status AT%I* : BOOL;

	ScreenCompactor_C101B_command AT%Q* : BOOL;

	ScreenCompactor_C101B_in : BOOL;
	ScreenCompactor_C101B_overload_error : BOOL;
	ScreenCompactor_C101B_incomplete_error : BOOL;
	ScreenCompactor_C101B_status_error : BOOL;
	ScreenCompactor_C101B_common_error : BOOL;
	ScreenCompactor_C101B_stop_error : BOOL;

	ScreenCompactor_C101B_overload_Filter : ErrorFilter;
	ScreenCompactor_C101B_incomplete_Filter : ErrorFilter;
	ScreenCompactor_C101B_status_Filter : ErrorFilter;
	ScreenCompactor_C101B_stop_Filter : ErrorFilter;

	ContinuousWaterSpray_XV102B_remote_mode AT%I* : BOOL;
	ContinuousWaterSpray_XV102B_overload AT%I* : BOOL;
	ContinuousWaterSpray_XV102B_incomplete AT%I* : BOOL;
	ContinuousWaterSpray_XV102B_status AT%I* : BOOL;

	ContinuousWaterSpray_XV102B_command AT%Q* : BOOL;

	ContinuousWaterSpray_XV102B_in : BOOL;
	ContinuousWaterSpray_XV102B_overload_error : BOOL;
	ContinuousWaterSpray_XV102B_incomplete_error : BOOL;
	ContinuousWaterSpray_XV102B_status_error : BOOL;
	ContinuousWaterSpray_XV102B_common_error : BOOL;
	ContinuousWaterSpray_XV102B_stop_error : BOOL;

	ContinuousWaterSpray_XV102B_overload_Filter : ErrorFilter;
	ContinuousWaterSpray_XV102B_incomplete_Filter : ErrorFilter;
	ContinuousWaterSpray_XV102B_status_Filter : ErrorFilter;
	ContinuousWaterSpray_XV102B_stop_Filter : ErrorFilter;

	WaterSprayOff1: TOF;
	WaterSprayOff2: TOF;
END_VAR
VAR (* helpers for the ST form of the networks *)
	_en57 : BOOL;
	_t57 : BOOL;
	_en85 : BOOL;
	_t85 : BOOL;
END_VAR
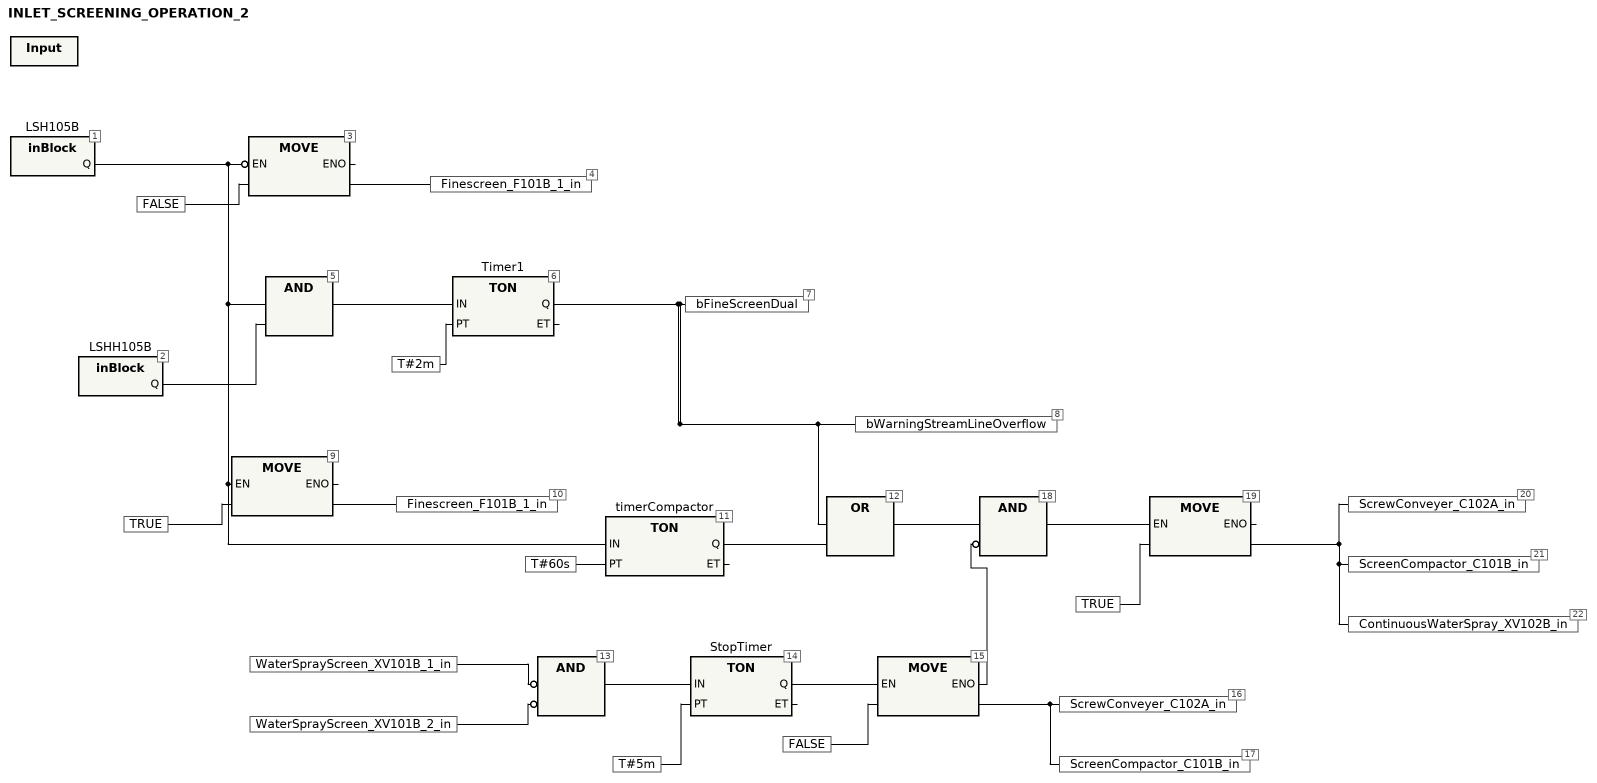
_CFC_ (* Continuous Function Chart, elements in execution order *)
#0 Input()
#1 LSH105B:inBlock()
#2 LSHH105B:inBlock()
#3 MOVE(EN: NOT #1.Q, FALSE)
#4 Finescreen_F101B_1_in <= #3
#5 AND(#1.Q, #2.Q)
#6 Timer1:TON(IN: #5, PT: T#2m)
#7 bFineScreenDual <= #6.Q
#8 bWarningStreamLineOverflow <= #6.Q
#9 MOVE(EN: #1.Q, TRUE)
#10 Finescreen_F101B_1_in <= #9
#11 timerCompactor:TON(IN: #1.Q, PT: T#60s)
#12 OR(#6.Q, #11.Q)
#13 AND(NOT WaterSprayScreen_XV101B_1_in, NOT WaterSprayScreen_XV101B_2_in)
#14 StopTimer:TON(IN: #13, PT: T#5m)
#15 MOVE(EN: #14.Q, FALSE)
#16 ScrewConveyer_C102A_in <= #15
#17 ScreenCompactor_C101B_in <= #15
#18 AND(#12, NOT #15.ENO)
#19 MOVE(EN: #18, TRUE)
#20 ScrewConveyer_C102A_in <= #19
#21 ScreenCompactor_C101B_in <= #19
#22 ContinuousWaterSpray_XV102B_in <= #19
_END_CFC_
(* the same logic as Structured Text *)
Input();
LSH105B();
LSHH105B();
IF NOT LSH105B.Q THEN Finescreen_F101B_1_in := FALSE; END_IF;
Timer1(IN := LSH105B.Q AND LSHH105B.Q, PT := T#2m);
bFineScreenDual := Timer1.Q;
bWarningStreamLineOverflow := Timer1.Q;
IF LSH105B.Q THEN Finescreen_F101B_1_in := TRUE; END_IF;
timerCompactor(IN := LSH105B.Q, PT := T#60s);
StopTimer(IN := NOT WaterSprayScreen_XV101B_1_in AND NOT WaterSprayScreen_XV101B_2_in, PT := T#5m);
_en57 := StopTimer.Q;
IF _en57 THEN _t57 := FALSE; END_IF;
IF _en57 THEN ScrewConveyer_C102A_in := _t57; END_IF;
IF _en57 THEN ScreenCompactor_C101B_in := _t57; END_IF;
_en85 := (Timer1.Q OR timerCompactor.Q) AND NOT _en57;
IF _en85 THEN _t85 := TRUE; END_IF;
IF _en85 THEN ScrewConveyer_C102A_in := _t85; END_IF;
IF _en85 THEN ScreenCompactor_C101B_in := _t85; END_IF;
IF _en85 THEN ContinuousWaterSpray_XV102B_in := _t85; END_IF;
END_PROGRAM
ACTION Input:
LSH105B( );
LSHH105B( );

Penstock_PS101B_1_command := Penstock_PS101B_1_in;
Penstock_PS101B_1_open_Filter(IN:=(NOT Penstock_PS101B_1_status AND Penstock_PS101B_1_in),PT:=T#10s, Q=>Penstock_PS101B_1_open_error);
Penstock_PS101B_1_close_Filter(IN:=( Penstock_PS101B_1_status AND NOT Penstock_PS101B_1_in),PT:=T#10s, Q=>Penstock_PS101B_1_close_error);

Penstock_PS101B_1_common_error := Penstock_PS101B_1_open_error OR Penstock_PS101B_1_close_error;


Penstock_PS101B_2_command := Penstock_PS101B_2_in;
Penstock_PS101B_2_open_Filter(IN:=(NOT Penstock_PS101B_2_status AND Penstock_PS101B_2_in),PT:=T#10s, Q=>Penstock_PS101B_2_open_error);
Penstock_PS101B_2_close_Filter(IN:=( Penstock_PS101B_2_status AND NOT Penstock_PS101B_2_in),PT:=T#10s, Q=>Penstock_PS101B_2_close_error);

Penstock_PS101B_2_common_error := Penstock_PS101B_2_open_error OR Penstock_PS101B_2_close_error;




Finescreen_F101B_1_overload_Filter(IN:=(Finescreen_F101B_1_overload AND Finescreen_F101B_1_in),PT:=T#2s,Q=>Finescreen_F101B_1_overload_error);
Finescreen_F101B_1_incomplete_Filter(IN:=(Finescreen_F101B_1_incomplete AND Finescreen_F101B_1_in),PT:=T#2s,Q=>Finescreen_F101B_1_incomplete_error);
Finescreen_F101B_1_status_Filter(IN:=(NOT Finescreen_F101B_1_status AND Finescreen_F101B_1_in),PT:=T#10s, Q=>Finescreen_F101B_1_status_error);
Finescreen_F101B_1_stop_Filter(IN:=( Finescreen_F101B_1_status AND NOT Finescreen_F101B_1_in),PT:=T#10s, Q=>Finescreen_F101B_1_stop_error);

Finescreen_F101B_1_common_error := Finescreen_F101B_1_overload_error OR Finescreen_F101B_1_incomplete_error OR Finescreen_F101B_1_status_error OR Finescreen_F101B_1_stop_error;


Finescreen_F101B_2_overload_Filter(IN:=(Finescreen_F101B_2_overload AND Finescreen_F101B_2_in),PT:=T#2s,Q=>Finescreen_F101B_2_overload_error);
Finescreen_F101B_2_incomplete_Filter(IN:=(Finescreen_F101B_2_incomplete AND Finescreen_F101B_2_in),PT:=T#2s,Q=>Finescreen_F101B_2_incomplete_error);
Finescreen_F101B_2_status_Filter(IN:=(NOT Finescreen_F101B_2_status AND Finescreen_F101B_2_in),PT:=T#10s, Q=>Finescreen_F101B_2_status_error);
Finescreen_F101B_2_stop_Filter(IN:=( Finescreen_F101B_2_status AND NOT Finescreen_F101B_2_in),PT:=T#10s, Q=>Finescreen_F101B_2_stop_error);

Finescreen_F101B_2_common_error := Finescreen_F101B_2_overload_error OR Finescreen_F101B_2_incomplete_error OR Finescreen_F101B_2_status_error OR Finescreen_F101B_2_stop_error;


FineScreen(
	ERROR1:=Finescreen_F101B_1_common_error ,
	ERROR2:=Finescreen_F101B_2_common_error ,
	IN1:= Finescreen_F101B_1_in,
	IN2:=Finescreen_F101B_2_in ,
	remote1:=Finescreen_F101B_1_remote_mode ,
	remote2:= Finescreen_F101B_2_remote_mode,
	Command1=>Finescreen_F101B_1_command ,
	Command2=>Finescreen_F101B_2_command );

IF bFineScreenDual THEN
	Finescreen_F101B_2_command := TRUE;
END_IF


Penstock_PS101B_1_in := Finescreen_F101B_1_command;
Penstock_PS101B_2_in := Finescreen_F101B_2_command;

WaterSprayOff1(IN:=Finescreen_F101B_1_command , PT:=T#2m , Q=>WaterSprayScreen_XV101B_1_in , ET=> );
WaterSprayOff2(IN:=Finescreen_F101B_2_command , PT:=T#2m , Q=>WaterSprayScreen_XV101B_2_in , ET=> );


WaterSprayScreen1(
	PT1:= T#1m,
	PT2:= T#5m,
	IN1:= WaterSprayScreen_XV101B_1_in,
	Command1=>WaterSprayScreen_XV101B_1_command );

WaterSprayScreen_XV101B_1_open_Filter(IN:=((NOT WaterSprayScreen_XV101B_1_open_status OR WaterSprayScreen_XV101B_1_close_status) AND WaterSprayScreen_XV101B_1_command),PT:=T#10s, Q=>WaterSprayScreen_XV101B_1_open_error);
WaterSprayScreen_XV101B_1_close_Filter(IN:=(( WaterSprayScreen_XV101B_1_open_status OR NOT WaterSprayScreen_XV101B_1_close_status) AND NOT WaterSprayScreen_XV101B_1_command),PT:=T#10s, Q=>WaterSprayScreen_XV101B_1_close_error);

WaterSprayScreen_XV101B_1_common_error := WaterSprayScreen_XV101B_1_open_error OR WaterSprayScreen_XV101B_1_close_error;


WaterSprayScreen2(
	PT1:= T#1m,
	PT2:= T#5m,
	IN1:= WaterSprayScreen_XV101B_2_in,
	Command1=>WaterSprayScreen_XV101B_2_command );

WaterSprayScreen_XV101B_2_open_Filter(IN:=((NOT WaterSprayScreen_XV101B_2_open_status OR WaterSprayScreen_XV101B_2_close_status) AND WaterSprayScreen_XV101B_2_in),PT:=T#10s, Q=>WaterSprayScreen_XV101B_2_open_error);
WaterSprayScreen_XV101B_2_close_Filter(IN:=((WaterSprayScreen_XV101B_2_open_status OR NOT WaterSprayScreen_XV101B_2_close_status) AND NOT WaterSprayScreen_XV101B_2_in),PT:=T#10s, Q=>WaterSprayScreen_XV101B_2_close_error);

WaterSprayScreen_XV101B_2_common_error := WaterSprayScreen_XV101B_2_open_error OR WaterSprayScreen_XV101B_2_close_error;


ScrewConveyer_C102A_command :=ScrewConveyer_C102A_in AND ScrewConveyer_C102A_remote_mode;
ScrewConveyer_C102A_overload_Filter(IN:=(ScrewConveyer_C102A_overload AND ScrewConveyer_C102A_in),PT:=T#2s,Q=>ScrewConveyer_C102A_overload_error);
ScrewConveyer_C102A_incomplete_Filter(IN:=(ScrewConveyer_C102A_incomplete AND ScrewConveyer_C102A_in),PT:=T#2s,Q=>ScrewConveyer_C102A_incomplete_error);
ScrewConveyer_C102A_status_Filter(IN:=(NOT ScrewConveyer_C102A_status AND ScrewConveyer_C102A_in),PT:=T#10s, Q=>ScrewConveyer_C102A_status_error);
ScrewConveyer_C102A_stop_Filter(IN:=( ScrewConveyer_C102A_status AND NOT ScrewConveyer_C102A_in),PT:=T#10s, Q=>ScrewConveyer_C102A_stop_error);

ScrewConveyer_C102A_common_error := ScrewConveyer_C102A_overload_error OR ScrewConveyer_C102A_incomplete_error OR ScrewConveyer_C102A_status_error OR ScrewConveyer_C102A_stop_error;


ScreenCompactor_C101B_command := ScreenCompactor_C101B_in OR ScreenCompactor_C101B_remote_mode;
ScreenCompactor_C101B_overload_Filter(IN:=(ScreenCompactor_C101B_overload AND ScreenCompactor_C101B_in),PT:=T#2s,Q=>ScreenCompactor_C101B_overload_error);
ScreenCompactor_C101B_incomplete_Filter(IN:=(ScreenCompactor_C101B_incomplete AND ScreenCompactor_C101B_in),PT:=T#2s,Q=>ScreenCompactor_C101B_incomplete_error);
ScreenCompactor_C101B_status_Filter(IN:=(NOT ScreenCompactor_C101B_status AND ScreenCompactor_C101B_in),PT:=T#10s, Q=>ScreenCompactor_C101B_status_error);
ScreenCompactor_C101B_stop_Filter(IN:=( ScreenCompactor_C101B_status AND NOT ScreenCompactor_C101B_in),PT:=T#10s, Q=>ScreenCompactor_C101B_stop_error);

ScreenCompactor_C101B_common_error := ScreenCompactor_C101B_overload_error OR ScreenCompactor_C101B_incomplete_error OR ScreenCompactor_C101B_status_error OR ScreenCompactor_C101B_stop_error;


ContinuousWaterSpray_XV102B_command := ContinuousWaterSpray_XV102B_in;
ContinuousWaterSpray_XV102B_overload_Filter(IN:=(ContinuousWaterSpray_XV102B_overload AND ContinuousWaterSpray_XV102B_in),PT:=T#2s,Q=>ContinuousWaterSpray_XV102B_overload_error);
ContinuousWaterSpray_XV102B_incomplete_Filter(IN:=(ContinuousWaterSpray_XV102B_incomplete AND ContinuousWaterSpray_XV102B_in),PT:=T#2s,Q=>ContinuousWaterSpray_XV102B_incomplete_error);
ContinuousWaterSpray_XV102B_status_Filter(IN:=(NOT ContinuousWaterSpray_XV102B_status AND ContinuousWaterSpray_XV102B_in),PT:=T#10s, Q=>ContinuousWaterSpray_XV102B_status_error);
ContinuousWaterSpray_XV102B_stop_Filter(IN:=( ContinuousWaterSpray_XV102B_status AND NOT ContinuousWaterSpray_XV102B_in),PT:=T#10s, Q=>ContinuousWaterSpray_XV102B_stop_error);

ContinuousWaterSpray_XV102B_common_error := ContinuousWaterSpray_XV102B_overload_error OR ContinuousWaterSpray_XV102B_incomplete_error OR ContinuousWaterSpray_XV102B_status_error OR ContinuousWaterSpray_XV102B_stop_error;
END_ACTION

(* POU GRIT_REMOVAL_OPERATION, CFC *)
PROGRAM GRIT_REMOVAL_OPERATION
VAR
	bGritClasifierOperation: BOOL;
	bSuctionValveOperation: BOOL;
	offGritClassifier: TON;

	GritAirBlower_B101A :Equipment_Dual_Timed;

	GritAirBlower_B101A_1_remote_mode AT%I* : BOOL;
	GritAirBlower_B101A_1_overload AT%I* : BOOL;
	GritAirBlower_B101A_1_incomplete AT%I* : BOOL;
	GritAirBlower_B101A_1_status AT%I* : BOOL;

	GritAirBlower_B101A_1_command AT%Q* : BOOL;

	GritAirBlower_B101A_1_in : BOOL;
	GritAirBlower_B101A_1_overload_error : BOOL;
	GritAirBlower_B101A_1_incomplete_error : BOOL;
	GritAirBlower_B101A_1_status_error : BOOL;
	GritAirBlower_B101A_1_common_error : BOOL;
	GritAirBlower_B101A_1_stop_error : BOOL;

	GritAirBlower_B101A_1_overload_Filter : ErrorFilter;
	GritAirBlower_B101A_1_incomplete_Filter : ErrorFilter;
	GritAirBlower_B101A_1_status_Filter : ErrorFilter;
	GritAirBlower_B101A_1_stop_Filter : ErrorFilter;



	GritAirBlower_B101A_2_remote_mode AT%I* : BOOL;
	GritAirBlower_B101A_2_overload AT%I* : BOOL;
	GritAirBlower_B101A_2_incomplete AT%I* : BOOL;
	GritAirBlower_B101A_2_status AT%I* : BOOL;

	GritAirBlower_B101A_2_command AT%Q* : BOOL;

	GritAirBlower_B101A_2_in : BOOL;
	GritAirBlower_B101A_2_overload_error : BOOL;
	GritAirBlower_B101A_2_incomplete_error : BOOL;
	GritAirBlower_B101A_2_status_error : BOOL;
	GritAirBlower_B101A_2_common_error : BOOL;
	GritAirBlower_B101A_2_stop_error : BOOL;

	GritAirBlower_B101A_2_overload_Filter : ErrorFilter;
	GritAirBlower_B101A_2_incomplete_Filter : ErrorFilter;
	GritAirBlower_B101A_2_status_Filter : ErrorFilter;
	GritAirBlower_B101A_2_stop_Filter : ErrorFilter;



	GritRemovalSuctionValve_XV100A_1_status AT%I* : BOOL;

	GritRemovalSuctionValve_XV100A_1_command AT%Q* : BOOL;

	GritRemovalSuctionValve_XV100A_1_in : BOOL;
	GritRemovalSuctionValve_XV100A_1_open_error : BOOL;
	GritRemovalSuctionValve_XV100A_1_common_error : BOOL;
	GritRemovalSuctionValve_XV100A_1_close_error : BOOL;

	GritRemovalSuctionValve_XV100A_1_open_Filter : ErrorFilter;
	GritRemovalSuctionValve_XV100A_1_close_Filter : ErrorFilter;



	GritRemovalSuctionValve_XV100A_2_status AT%I* : BOOL;

	GritRemovalSuctionValve_XV100A_2_command AT%Q* : BOOL;

	GritRemovalSuctionValve_XV100A_2_in : BOOL;
	GritRemovalSuctionValve_XV100A_2_open_error : BOOL;
	GritRemovalSuctionValve_XV100A_2_common_error : BOOL;
	GritRemovalSuctionValve_XV100A_2_close_error : BOOL;

	GritRemovalSuctionValve_XV100A_2_open_Filter : ErrorFilter;
	GritRemovalSuctionValve_XV100A_2_close_Filter : ErrorFilter;


	GritRemovalSuctionValve_XV100B_1_status AT%I* : BOOL;

	GritRemovalSuctionValve_XV100B_1_command AT%Q* : BOOL;

	GritRemovalSuctionValve_XV100B_1_in : BOOL;
	GritRemovalSuctionValve_XV100B_1_open_error : BOOL;
	GritRemovalSuctionValve_XV100B_1_common_error : BOOL;
	GritRemovalSuctionValve_XV100B_1_close_error : BOOL;

	GritRemovalSuctionValve_XV100B_1_open_Filter : ErrorFilter;
	GritRemovalSuctionValve_XV100B_1_close_Filter : ErrorFilter;


	GritRemovalSuctionValve_XV100B_2_status AT%I* : BOOL;

	GritRemovalSuctionValve_XV100B_2_command AT%Q* : BOOL;

	GritRemovalSuctionValve_XV100B_2_in : BOOL;
	GritRemovalSuctionValve_XV100B_2_open_error : BOOL;
	GritRemovalSuctionValve_XV100B_2_common_error : BOOL;
	GritRemovalSuctionValve_XV100B_2_close_error : BOOL;

	GritRemovalSuctionValve_XV100B_2_open_Filter : ErrorFilter;
	GritRemovalSuctionValve_XV100B_2_close_Filter : ErrorFilter;


	GritClassifier_C103A_remote_mode AT%I* : BOOL;
	GritClassifier_C103A_overload AT%I* : BOOL;
	GritClassifier_C103A_incomplete AT%I* : BOOL;
	GritClassifier_C103A_status AT%I* : BOOL;

	GritClassifier_C103A_command AT%Q* : BOOL;

	GritClassifier_C103A_in : BOOL;
	GritClassifier_C103A_overload_error : BOOL;
	GritClassifier_C103A_incomplete_error : BOOL;
	GritClassifier_C103A_status_error : BOOL;
	GritClassifier_C103A_common_error : BOOL;
	GritClassifier_C103A_stop_error : BOOL;

	GritClassifier_C103A_overload_Filter : ErrorFilter;
	GritClassifier_C103A_incomplete_Filter : ErrorFilter;
	GritClassifier_C103A_status_Filter : ErrorFilter;
	GritClassifier_C103A_stop_Filter : ErrorFilter;



	GritClassifier_C103B_remote_mode AT%I* : BOOL;
	GritClassifier_C103B_overload AT%I* : BOOL;
	GritClassifier_C103B_incomplete AT%I* : BOOL;
	GritClassifier_C103B_status AT%I* : BOOL;

	GritClassifier_C103B_command AT%Q* : BOOL;

	GritClassifier_C103B_in : BOOL;
	GritClassifier_C103B_overload_error : BOOL;
	GritClassifier_C103B_incomplete_error : BOOL;
	GritClassifier_C103B_status_error : BOOL;
	GritClassifier_C103B_common_error : BOOL;
	GritClassifier_C103B_stop_error : BOOL;

	GritClassifier_C103B_overload_Filter : ErrorFilter;
	GritClassifier_C103B_incomplete_Filter : ErrorFilter;
	GritClassifier_C103B_status_Filter : ErrorFilter;
	GritClassifier_C103B_stop_Filter : ErrorFilter;


	B101AdutyStart: BOOL;
	B101AstandbyStart: BOOL;
END_VAR
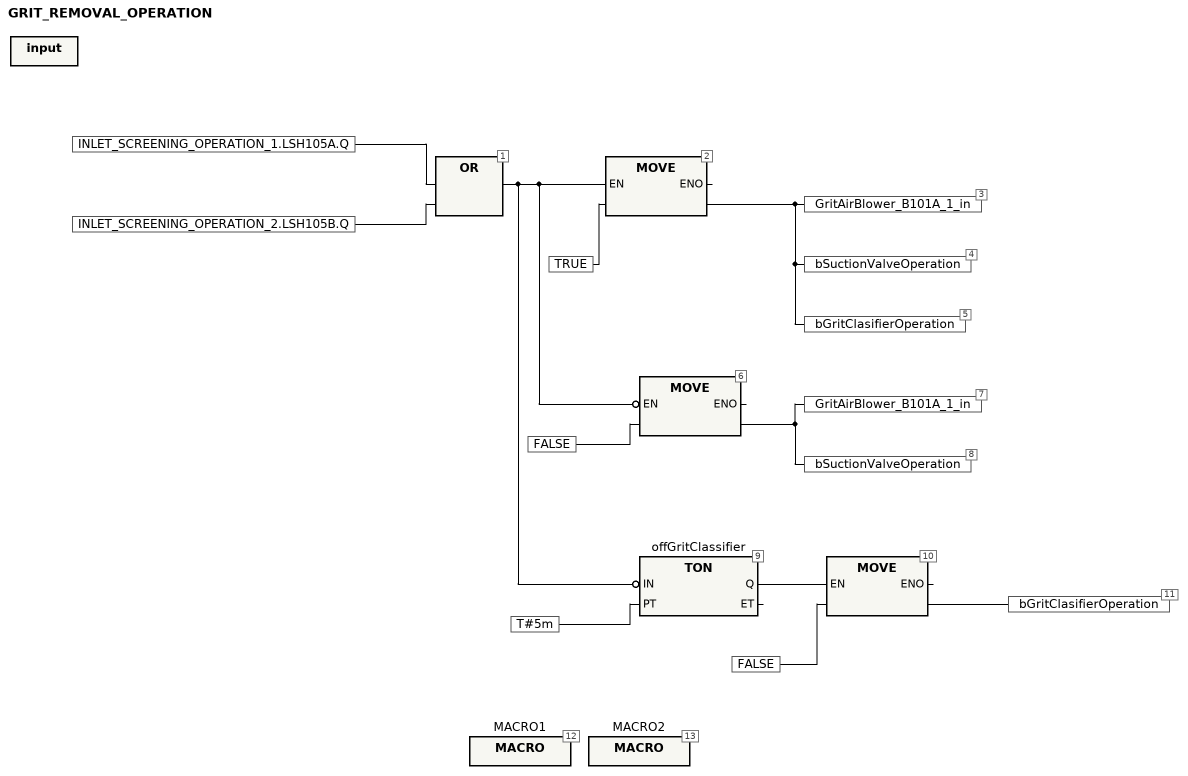
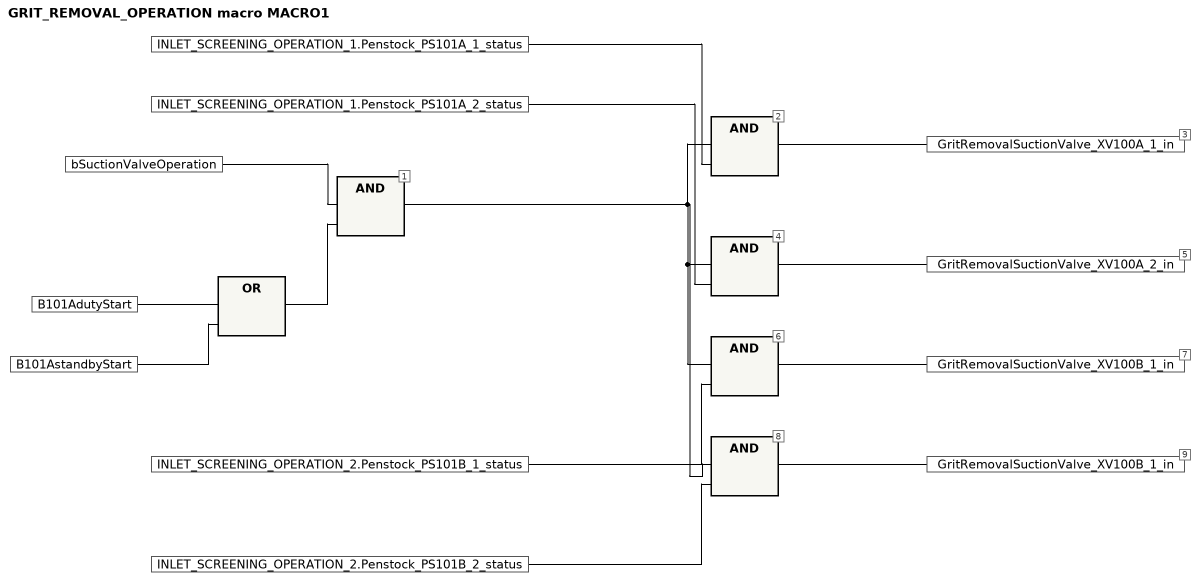
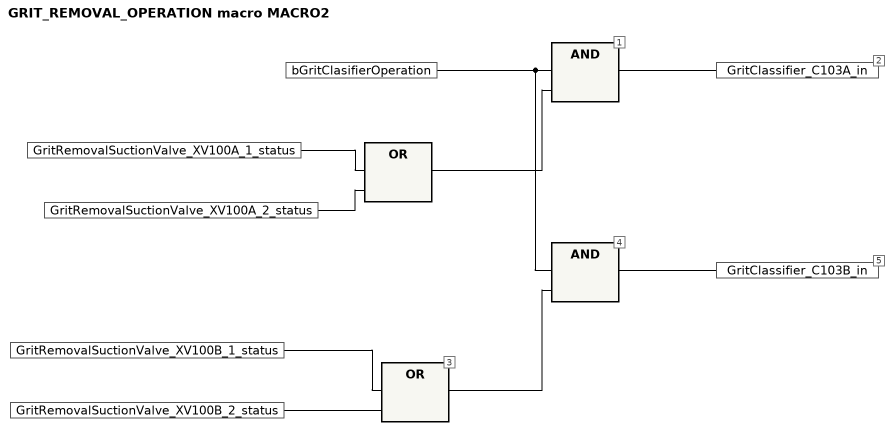
_CFC_ (* Continuous Function Chart, elements in execution order *)
#0 input()
#1 OR(INLET_SCREENING_OPERATION_1.LSH105A.Q, INLET_SCREENING_OPERATION_2.LSH105B.Q)
#2 MOVE(EN: #1, TRUE)
#3 GritAirBlower_B101A_1_in <= #2
#4 bSuctionValveOperation <= #2
#5 bGritClasifierOperation <= #2
#6 MOVE(EN: NOT #1, FALSE)
#7 GritAirBlower_B101A_1_in <= #6
#8 bSuctionValveOperation <= #6
#9 offGritClassifier:TON(IN: NOT #1, PT: T#5m)
#10 MOVE(EN: #9.Q, FALSE)
#11 bGritClasifierOperation <= #10
#12 MACRO MACRO1()
	#13 OR(B101AdutyStart, B101AstandbyStart)
	#14 AND(bSuctionValveOperation, #13)
	#15 AND(#14, INLET_SCREENING_OPERATION_1.Penstock_PS101A_1_status)
	#16 GritRemovalSuctionValve_XV100A_1_in <= #15
	#17 AND(#14, INLET_SCREENING_OPERATION_1.Penstock_PS101A_2_status)
	#18 GritRemovalSuctionValve_XV100A_2_in <= #17
	#19 AND(#14, INLET_SCREENING_OPERATION_2.Penstock_PS101B_1_status)
	#20 GritRemovalSuctionValve_XV100B_1_in <= #19
	#21 AND(#14, INLET_SCREENING_OPERATION_2.Penstock_PS101B_2_status)
	#22 GritRemovalSuctionValve_XV100B_1_in <= #21
END_MACRO
#23 MACRO MACRO2()
	#24 OR(GritRemovalSuctionValve_XV100A_1_status, GritRemovalSuctionValve_XV100A_2_status)
	#25 AND(bGritClasifierOperation, #24)
	#26 GritClassifier_C103A_in <= #25
	#27 OR(GritRemovalSuctionValve_XV100B_1_status, GritRemovalSuctionValve_XV100B_2_status)
	#28 AND(bGritClasifierOperation, #27)
	#29 GritClassifier_C103B_in <= #28
END_MACRO
_END_CFC_
END_PROGRAM
ACTION input:
GritAirBlower_B101A_1_overload_Filter(IN:=(GritAirBlower_B101A_1_overload AND GritAirBlower_B101A_1_in),PT:=T#2s,Q=>GritAirBlower_B101A_1_overload_error);
GritAirBlower_B101A_1_incomplete_Filter(IN:=(GritAirBlower_B101A_1_incomplete AND GritAirBlower_B101A_1_in),PT:=T#2s,Q=>GritAirBlower_B101A_1_incomplete_error);
GritAirBlower_B101A_1_status_Filter(IN:=(NOT GritAirBlower_B101A_1_status AND GritAirBlower_B101A_1_in),PT:=T#10s, Q=>GritAirBlower_B101A_1_status_error);
GritAirBlower_B101A_1_stop_Filter(IN:=( GritAirBlower_B101A_1_status AND NOT GritAirBlower_B101A_1_in),PT:=T#10s, Q=>GritAirBlower_B101A_1_stop_error);

GritAirBlower_B101A_1_common_error := GritAirBlower_B101A_1_overload_error OR GritAirBlower_B101A_1_incomplete_error OR GritAirBlower_B101A_1_status_error OR GritAirBlower_B101A_1_stop_error;

GritAirBlower_B101A_2_overload_Filter(IN:=(GritAirBlower_B101A_2_overload AND GritAirBlower_B101A_2_in),PT:=T#2s,Q=>GritAirBlower_B101A_2_overload_error);
GritAirBlower_B101A_2_incomplete_Filter(IN:=(GritAirBlower_B101A_2_incomplete AND GritAirBlower_B101A_2_in),PT:=T#2s,Q=>GritAirBlower_B101A_2_incomplete_error);
GritAirBlower_B101A_2_status_Filter(IN:=(NOT GritAirBlower_B101A_2_status AND GritAirBlower_B101A_2_in),PT:=T#10s, Q=>GritAirBlower_B101A_2_status_error);
GritAirBlower_B101A_2_stop_Filter(IN:=( GritAirBlower_B101A_2_status AND NOT GritAirBlower_B101A_2_in),PT:=T#10s, Q=>GritAirBlower_B101A_2_stop_error);

GritAirBlower_B101A_2_common_error := GritAirBlower_B101A_2_overload_error OR GritAirBlower_B101A_2_incomplete_error OR GritAirBlower_B101A_2_status_error OR GritAirBlower_B101A_2_stop_error;

GritAirBlower_B101A(
	ERROR1:= GritAirBlower_B101A_1_common_error,
	ERROR2:= GritAirBlower_B101A_2_common_error,
	remote1:= GritAirBlower_B101A_1_remote_mode,
	remote2:= GritAirBlower_B101A_2_remote_mode,
	PT1:=T#60m ,
	PT2:= T#60m,
	IN1:=GritAirBlower_B101A_1_in ,
	IN2:= GritAirBlower_B101A_2_in,
	Command1=>GritAirBlower_B101A_1_command ,
	Command2=>GritAirBlower_B101A_2_command );


GritRemovalSuctionValve_XV100A_1_command := GritRemovalSuctionValve_XV100A_1_in;
GritRemovalSuctionValve_XV100A_1_open_Filter(IN:=(NOT GritRemovalSuctionValve_XV100A_1_status AND GritRemovalSuctionValve_XV100A_1_in),PT:=T#10s, Q=>GritRemovalSuctionValve_XV100A_1_open_error);
GritRemovalSuctionValve_XV100A_1_close_Filter(IN:=( GritRemovalSuctionValve_XV100A_1_status AND NOT GritRemovalSuctionValve_XV100A_1_in),PT:=T#10s, Q=>GritRemovalSuctionValve_XV100A_1_close_error);

GritRemovalSuctionValve_XV100A_1_common_error := GritRemovalSuctionValve_XV100A_1_open_error OR GritRemovalSuctionValve_XV100A_1_close_error;


GritRemovalSuctionValve_XV100A_2_command := GritRemovalSuctionValve_XV100A_2_in;
GritRemovalSuctionValve_XV100A_2_open_Filter(IN:=(NOT GritRemovalSuctionValve_XV100A_2_status AND GritRemovalSuctionValve_XV100A_2_in),PT:=T#10s, Q=>GritRemovalSuctionValve_XV100A_2_open_error);
GritRemovalSuctionValve_XV100A_2_close_Filter(IN:=( GritRemovalSuctionValve_XV100A_2_status AND NOT GritRemovalSuctionValve_XV100A_2_in),PT:=T#10s, Q=>GritRemovalSuctionValve_XV100A_2_close_error);

GritRemovalSuctionValve_XV100A_2_common_error := GritRemovalSuctionValve_XV100A_2_open_error OR GritRemovalSuctionValve_XV100A_2_close_error;




GritRemovalSuctionValve_XV100B_1_command := GritRemovalSuctionValve_XV100B_1_in;
GritRemovalSuctionValve_XV100B_1_open_Filter(IN:=(NOT GritRemovalSuctionValve_XV100B_1_status AND GritRemovalSuctionValve_XV100B_1_in),PT:=T#10s, Q=>GritRemovalSuctionValve_XV100B_1_open_error);
GritRemovalSuctionValve_XV100B_1_close_Filter(IN:=( GritRemovalSuctionValve_XV100B_1_status AND NOT GritRemovalSuctionValve_XV100B_1_in),PT:=T#10s, Q=>GritRemovalSuctionValve_XV100B_1_close_error);

GritRemovalSuctionValve_XV100B_1_common_error := GritRemovalSuctionValve_XV100B_1_open_error OR GritRemovalSuctionValve_XV100B_1_close_error;



GritRemovalSuctionValve_XV100B_2_command := GritRemovalSuctionValve_XV100B_2_in;
GritRemovalSuctionValve_XV100B_2_open_Filter(IN:=(NOT GritRemovalSuctionValve_XV100B_2_status AND GritRemovalSuctionValve_XV100B_2_in),PT:=T#10s, Q=>GritRemovalSuctionValve_XV100B_2_open_error);
GritRemovalSuctionValve_XV100B_2_close_Filter(IN:=( GritRemovalSuctionValve_XV100B_2_status AND NOT GritRemovalSuctionValve_XV100B_2_in),PT:=T#10s, Q=>GritRemovalSuctionValve_XV100B_2_close_error);

GritRemovalSuctionValve_XV100B_2_common_error := GritRemovalSuctionValve_XV100B_2_open_error OR GritRemovalSuctionValve_XV100B_2_close_error;



GritClassifier_C103A_command := GritClassifier_C103A_in AND GritClassifier_C103A_remote_mode;
GritClassifier_C103A_overload_Filter(IN:=(GritClassifier_C103A_overload AND GritClassifier_C103A_in),PT:=T#2s,Q=>GritClassifier_C103A_overload_error);
GritClassifier_C103A_incomplete_Filter(IN:=(GritClassifier_C103A_incomplete AND GritClassifier_C103A_in),PT:=T#2s,Q=>GritClassifier_C103A_incomplete_error);
GritClassifier_C103A_status_Filter(IN:=(NOT GritClassifier_C103A_status AND GritClassifier_C103A_in),PT:=T#10s, Q=>GritClassifier_C103A_status_error);
GritClassifier_C103A_stop_Filter(IN:=( GritClassifier_C103A_status AND NOT GritClassifier_C103A_in),PT:=T#10s, Q=>GritClassifier_C103A_stop_error);

GritClassifier_C103A_common_error := GritClassifier_C103A_overload_error OR GritClassifier_C103A_incomplete_error OR GritClassifier_C103A_status_error OR GritClassifier_C103A_stop_error;



GritClassifier_C103B_command := GritClassifier_C103B_in AND GritClassifier_C103B_remote_mode;
GritClassifier_C103B_overload_Filter(IN:=(GritClassifier_C103B_overload AND GritClassifier_C103B_in),PT:=T#2s,Q=>GritClassifier_C103B_overload_error);
GritClassifier_C103B_incomplete_Filter(IN:=(GritClassifier_C103B_incomplete AND GritClassifier_C103B_in),PT:=T#2s,Q=>GritClassifier_C103B_incomplete_error);
GritClassifier_C103B_status_Filter(IN:=(NOT GritClassifier_C103B_status AND GritClassifier_C103B_in),PT:=T#10s, Q=>GritClassifier_C103B_status_error);
GritClassifier_C103B_stop_Filter(IN:=( GritClassifier_C103B_status AND NOT GritClassifier_C103B_in),PT:=T#10s, Q=>GritClassifier_C103B_stop_error);

GritClassifier_C103B_common_error := GritClassifier_C103B_overload_error OR GritClassifier_C103B_incomplete_error OR GritClassifier_C103B_status_error OR GritClassifier_C103B_stop_error;
END_ACTION

(* POU module/Equipment_Dual_Timed, ST *)
FUNCTION_BLOCK Equipment_Dual_Timed
VAR_INPUT
	ERROR1 : BOOL;
	ERROR2 : BOOL;
	remote1 : BOOL;
	remote2 : BOOL;
	PT1: TIME;
	PT2: TIME;
END_VAR
VAR_OUTPUT
	Command1 : BOOL;
	Command2 : BOOL;
END_VAR
VAR_IN_OUT
	IN1 : BOOL;
	IN2 : BOOL;
END_VAR
VAR
	timer1: TP;
	timer2: TP;
	step: INT;
END_VAR
CASE step OF
0:
	Command1 := IN1 AND remote1;
	timer1(IN:= IN1 AND remote1, PT := PT1);
	IF ERROR1 THEN
		step := 10;
		timer1(IN:= FALSE, PT := PT1);
	ELSIF timer1.Q THEN
		command1 := FALSE;
		step := 10;
		timer1(IN:= FALSE, PT := PT1);
	END_IF
10:
	IN2 := IN1;
	Command2 := IN2 AND remote2;
	timer2(IN:=IN2 AND remote2,PT:=PT2);
	IF ERROR2 THEN
		step := 0;
		timer2(IN:=FALSE,PT:=PT2);
	ELSIF timer2.Q THEN
		Command2 := FALSE;
		IN2 := FALSE;
		timer2(IN:=FALSE,PT:=PT2);
		step := 0;
	END_IF
END_CASE
END_FUNCTION_BLOCK

(* POU REUSE_WATER_SYSTEM, CFC *)
PROGRAM REUSE_WATER_SYSTEM
VAR

	LSH405 : inBlock;
	LSL308A : inBlock;
	LSH308A : inBlock;
	FSL101:inBlock;
	PSL411 AT%I* : INT;
	PSL412 AT%I*: BOOL;
	bTriggerNegativePressure AT%I*: BOOL;
	bTriggerPositivePressure AT%I*: BOOL;
	rWaterPressureSensor:REAL;

	bPumpSequence: BOOL;
	bVacumPrimingOperation: BOOL;
	bOverrideON: BOOL;
	bOverrideOFF: BOOL;

	bWarningWaterPressureHigh: BOOL;
	bWarning_PrimingNoWater: BOOL;

	bSolenoidValve: BOOL;
	bVacumPumDuty: BOOL;
	bJokeyPump: BOOL;
	bLeadPumpAB: BOOL;
	bLeadPumpCD: BOOL;
	bJokeyPumpInternalOff: BOOL;

	WaitToFill: TON;
	TOverrideON: TON;
	TOverrideOFF: TON;
	Lower_3_5_timer: TON;


	SolenoidValve_XV102_status AT%I* : BOOL;

	SolenoidValve_XV102_command AT%Q* : BOOL;

	SolenoidValve_XV102_in : BOOL;
	SolenoidValve_XV102_open_error : BOOL;
	SolenoidValve_XV102_common_error : BOOL;
	SolenoidValve_XV102_close_error : BOOL;

	SolenoidValve_XV102_open_Filter : ErrorFilter;
	SolenoidValve_XV102_close_Filter : ErrorFilter;


	VacummPump_P403_A_remote_mode AT%I* : BOOL;
	VacummPump_P403_A_overload AT%I* : BOOL;
	VacummPump_P403_A_incomplete AT%I* : BOOL;
	VacummPump_P403_A_status AT%I* : BOOL;

	VacummPump_P403_A_command AT%Q* : BOOL;

	VacummPump_P403_A_in : BOOL;
	VacummPump_P403_A_overload_error : BOOL;
	VacummPump_P403_A_incomplete_error : BOOL;
	VacummPump_P403_A_status_error : BOOL;
	VacummPump_P403_A_common_error : BOOL;
	VacummPump_P403_A_stop_error : BOOL;

	VacummPump_P403_A_overload_Filter : ErrorFilter;
	VacummPump_P403_A_incomplete_Filter : ErrorFilter;
	VacummPump_P403_A_status_Filter : ErrorFilter;
	VacummPump_P403_A_stop_Filter : ErrorFilter;


	VacummPump_P403_B_remote_mode AT%I* : BOOL;
	VacummPump_P403_B_overload AT%I* : BOOL;
	VacummPump_P403_B_incomplete AT%I* : BOOL;
	VacummPump_P403_B_status AT%I* : BOOL;

	VacummPump_P403_B_command AT%Q* : BOOL;

	VacummPump_P403_B_in : BOOL;
	VacummPump_P403_B_overload_error : BOOL;
	VacummPump_P403_B_incomplete_error : BOOL;
	VacummPump_P403_B_status_error : BOOL;
	VacummPump_P403_B_common_error : BOOL;
	VacummPump_P403_B_stop_error : BOOL;

	VacummPump_P403_B_overload_Filter : ErrorFilter;
	VacummPump_P403_B_incomplete_Filter : ErrorFilter;
	VacummPump_P403_B_status_Filter : ErrorFilter;
	VacummPump_P403_B_stop_Filter : ErrorFilter;

	VacummPump_P403 :Equipment_Dual;


	JockeyPump_P402_A_remote_mode AT%I* : BOOL;
	JockeyPump_P402_A_overload AT%I* : BOOL;
	JockeyPump_P402_A_incomplete AT%I* : BOOL;
	JockeyPump_P402_A_status AT%I* : BOOL;

	JockeyPump_P402_A_command AT%Q* : BOOL;

	JockeyPump_P402_A_in : BOOL;
	JockeyPump_P402_A_overload_error : BOOL;
	JockeyPump_P402_A_incomplete_error : BOOL;
	JockeyPump_P402_A_status_error : BOOL;
	JockeyPump_P402_A_common_error : BOOL;
	JockeyPump_P402_A_stop_error : BOOL;

	JockeyPump_P402_A_overload_Filter : ErrorFilter;
	JockeyPump_P402_A_incomplete_Filter : ErrorFilter;
	JockeyPump_P402_A_status_Filter : ErrorFilter;
	JockeyPump_P402_A_stop_Filter : ErrorFilter;



	JockeyPump_P402_B_remote_mode AT%I* : BOOL;
	JockeyPump_P402_B_overload AT%I* : BOOL;
	JockeyPump_P402_B_incomplete AT%I* : BOOL;
	JockeyPump_P402_B_status AT%I* : BOOL;

	JockeyPump_P402_B_command AT%Q* : BOOL;

	JockeyPump_P402_B_in : BOOL;
	JockeyPump_P402_B_overload_error : BOOL;
	JockeyPump_P402_B_incomplete_error : BOOL;
	JockeyPump_P402_B_status_error : BOOL;
	JockeyPump_P402_B_common_error : BOOL;
	JockeyPump_P402_B_stop_error : BOOL;

	JockeyPump_P402_B_overload_Filter : ErrorFilter;
	JockeyPump_P402_B_incomplete_Filter : ErrorFilter;
	JockeyPump_P402_B_status_Filter : ErrorFilter;
	JockeyPump_P402_B_stop_Filter : ErrorFilter;

	JockeyPump_P402:Equipment_Dual;


	LeadPump_P401_A_remote_mode AT%I* : BOOL;
	LeadPump_P401_A_overload AT%I* : BOOL;
	LeadPump_P401_A_incomplete AT%I* : BOOL;
	LeadPump_P401_A_status AT%I* : BOOL;

	LeadPump_P401_A_command AT%Q* : BOOL;

	LeadPump_P401_A_in : BOOL;
	LeadPump_P401_A_overload_error : BOOL;
	LeadPump_P401_A_incomplete_error : BOOL;
	LeadPump_P401_A_status_error : BOOL;
	LeadPump_P401_A_common_error : BOOL;
	LeadPump_P401_A_stop_error : BOOL;

	LeadPump_P401_A_overload_Filter : ErrorFilter;
	LeadPump_P401_A_incomplete_Filter : ErrorFilter;
	LeadPump_P401_A_status_Filter : ErrorFilter;
	LeadPump_P401_A_stop_Filter : ErrorFilter;

	LeadPump_P401_B_remote_mode AT%I* : BOOL;
	LeadPump_P401_B_overload AT%I* : BOOL;
	LeadPump_P401_B_incomplete AT%I* : BOOL;
	LeadPump_P401_B_status AT%I* : BOOL;

	LeadPump_P401_B_command AT%Q* : BOOL;

	LeadPump_P401_B_in : BOOL;
	LeadPump_P401_B_overload_error : BOOL;
	LeadPump_P401_B_incomplete_error : BOOL;
	LeadPump_P401_B_status_error : BOOL;
	LeadPump_P401_B_common_error : BOOL;
	LeadPump_P401_B_stop_error : BOOL;

	LeadPump_P401_B_overload_Filter : ErrorFilter;
	LeadPump_P401_B_incomplete_Filter : ErrorFilter;
	LeadPump_P401_B_status_Filter : ErrorFilter;
	LeadPump_P401_B_stop_Filter : ErrorFilter;


	LeadPump_P401_C_remote_mode AT%I* : BOOL;
	LeadPump_P401_C_overload AT%I* : BOOL;
	LeadPump_P401_C_incomplete AT%I* : BOOL;
	LeadPump_P401_C_status AT%I* : BOOL;

	LeadPump_P401_C_command AT%Q* : BOOL;

	LeadPump_P401_C_in : BOOL;
	LeadPump_P401_C_overload_error : BOOL;
	LeadPump_P401_C_incomplete_error : BOOL;
	LeadPump_P401_C_status_error : BOOL;
	LeadPump_P401_C_common_error : BOOL;
	LeadPump_P401_C_stop_error : BOOL;

	LeadPump_P401_C_overload_Filter : ErrorFilter;
	LeadPump_P401_C_incomplete_Filter : ErrorFilter;
	LeadPump_P401_C_status_Filter : ErrorFilter;
	LeadPump_P401_C_stop_Filter : ErrorFilter;


	LeadPump_P401_D_remote_mode AT%I* : BOOL;
	LeadPump_P401_D_overload AT%I* : BOOL;
	LeadPump_P401_D_incomplete AT%I* : BOOL;
	LeadPump_P401_D_status AT%I* : BOOL;

	LeadPump_P401_D_command AT%Q* : BOOL;

	LeadPump_P401_D_in : BOOL;
	LeadPump_P401_D_overload_error : BOOL;
	LeadPump_P401_D_incomplete_error : BOOL;
	LeadPump_P401_D_status_error : BOOL;
	LeadPump_P401_D_common_error : BOOL;
	LeadPump_P401_D_stop_error : BOOL;

	LeadPump_P401_D_overload_Filter : ErrorFilter;
	LeadPump_P401_D_incomplete_Filter : ErrorFilter;
	LeadPump_P401_D_status_Filter : ErrorFilter;
	LeadPump_P401_D_stop_Filter : ErrorFilter;

	LeadPump_P401_A :Equipment_Single;
	LeadPump_P401_B :Equipment_Single;
	LeadPump_P401_C :Equipment_Single;
	LeadPump_P401_D :Equipment_Single;


END_VAR
VAR (* helpers for the ST form of the networks *)
	_t23 : BOOL;
	_t1 : BOOL;
	_t10 : BOOL;
	_t4 : BOOL;
	_t109 : BOOL;
	_t44 : BOOL;
	_en56 : BOOL;
	_en89 : BOOL;
	_t102 : BOOL;
	_t101 : BOOL;
	_t49 : BOOL;
	_t56 : BOOL;
	_t62 : BOOL;
	_en65 : BOOL;
	_t65 : BOOL;
	_t68 : BOOL;
	_t73 : BOOL;
	_t77 : BOOL;
	_en78 : BOOL;
	_t78 : BOOL;
	_t89 : BOOL;
	_t88 : BOOL;
	_t97 : BOOL;
END_VAR
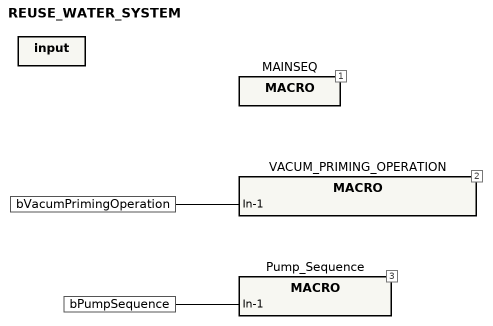
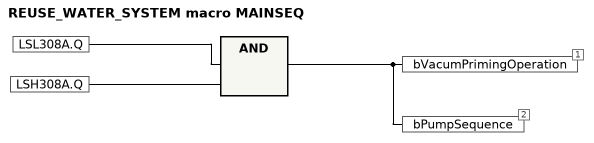
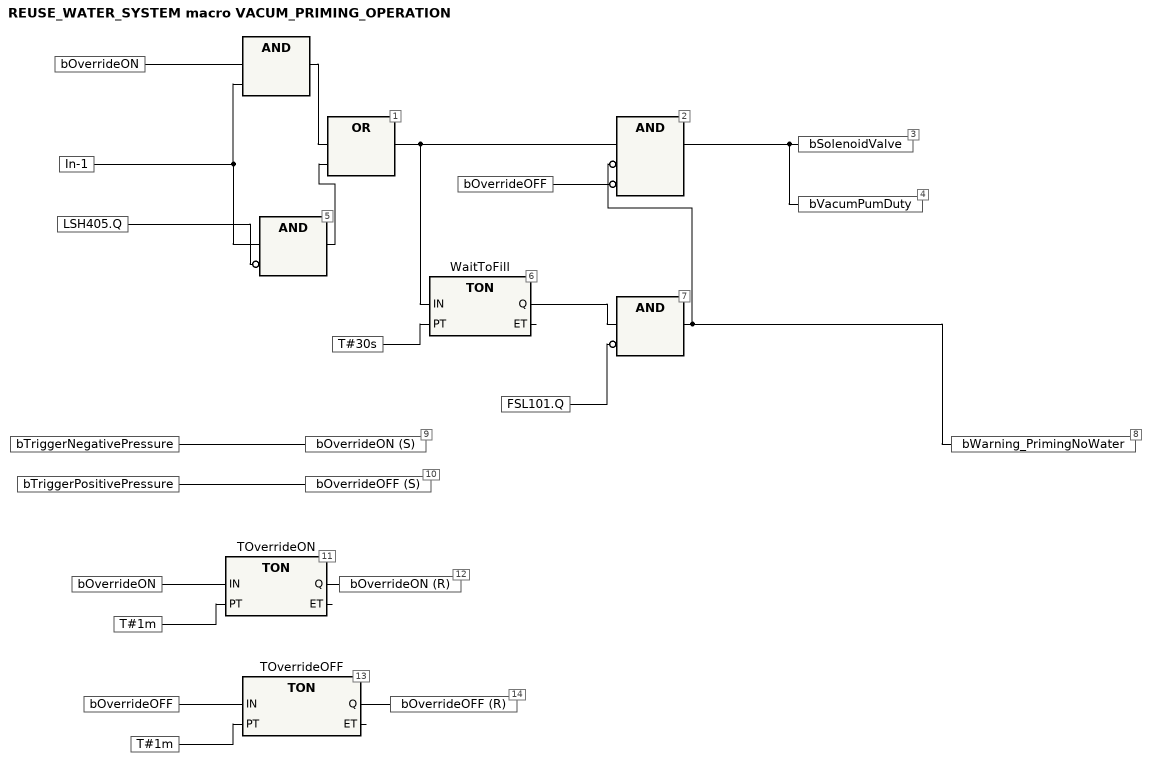
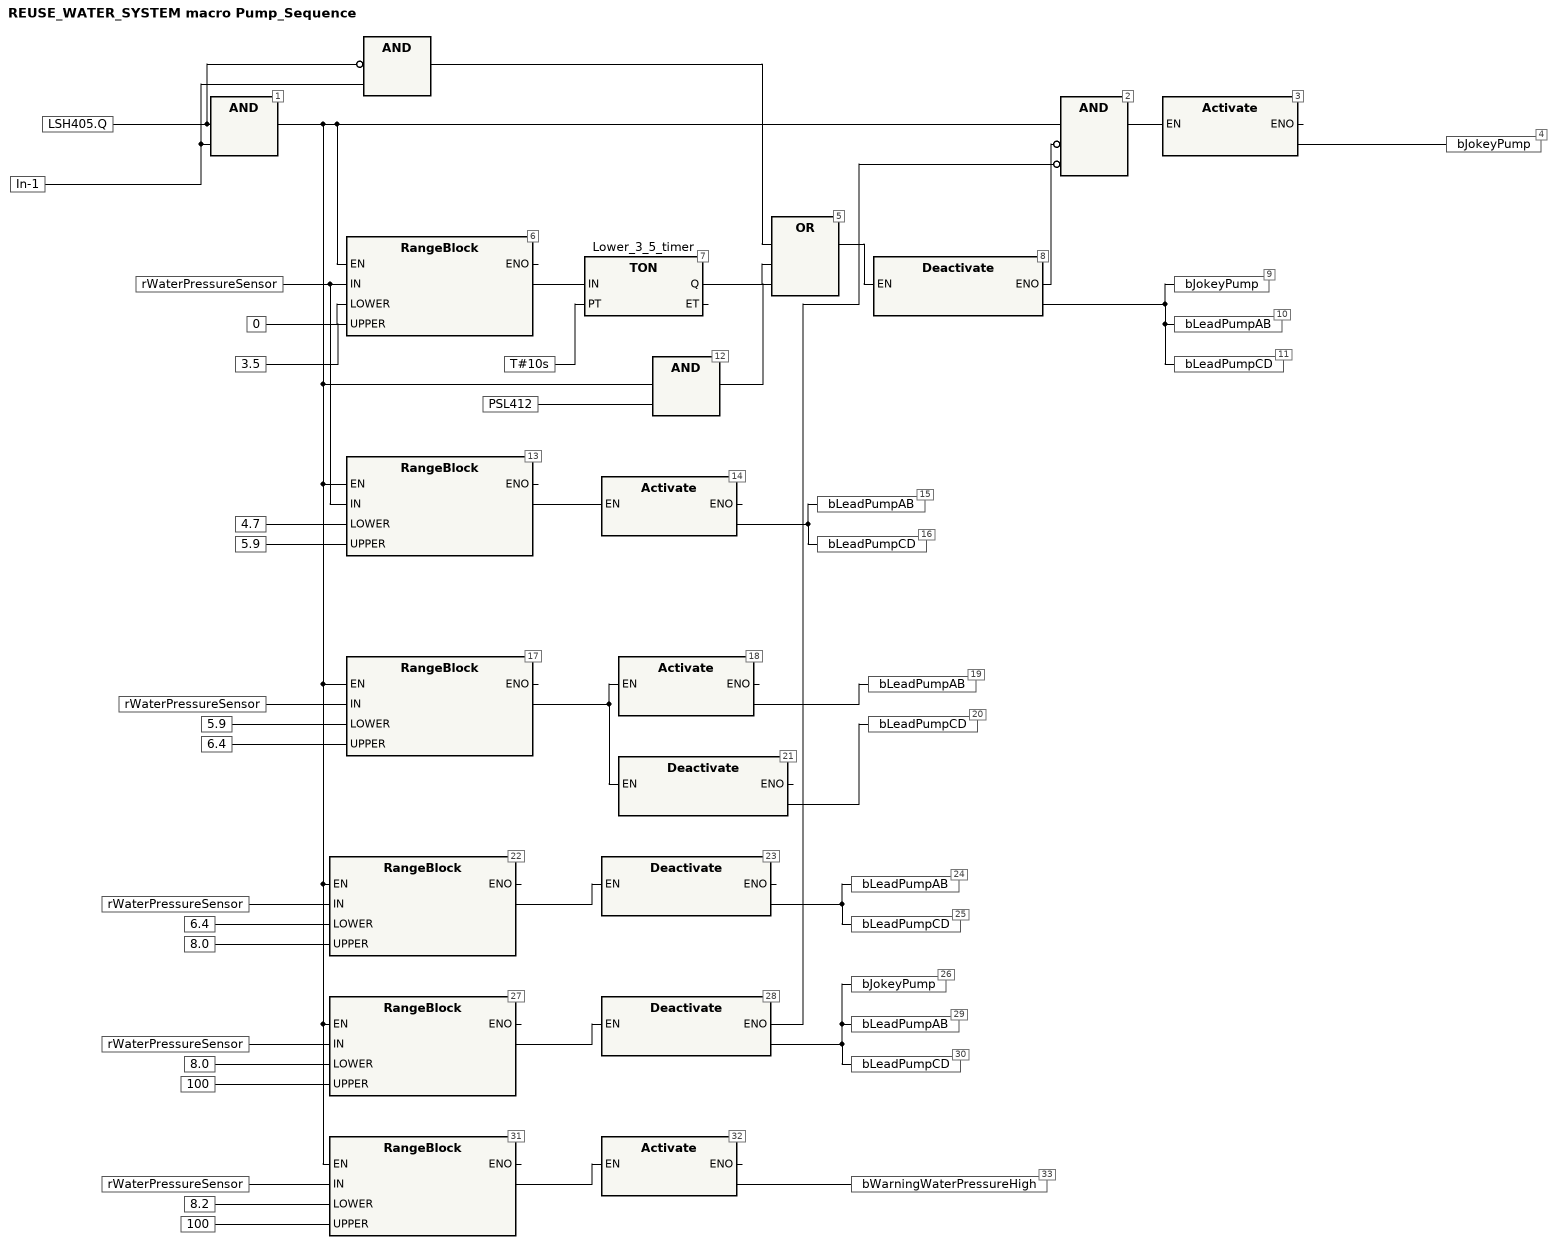
_CFC_ (* Continuous Function Chart, elements in execution order *)
#0 input()
#1 MACRO MAINSEQ()
	#2 AND(LSL308A.Q, LSH308A.Q)
	#3 bVacumPrimingOperation <= #2
	#4 bPumpSequence <= #2
END_MACRO
#5 MACRO VACUM_PRIMING_OPERATION(pin 1 "In-1": bVacumPrimingOperation)
	#6 AND(bOverrideON, pin 1)
	#7 OR(#6, #11)
	#8 AND(#7, NOT #13, NOT bOverrideOFF)
	#9 bSolenoidValve <= #8
	#10 bVacumPumDuty <= #8
	#11 AND(pin 1, NOT LSH405.Q)
	#12 WaitToFill:TON(IN: #7, PT: T#30s)
	#13 AND(#12.Q, NOT FSL101.Q)
	#14 bWarning_PrimingNoWater <= #13
	#15 S bOverrideON <= bTriggerNegativePressure
	#16 S bOverrideOFF <= bTriggerPositivePressure
	#17 TOverrideON:TON(IN: bOverrideON, PT: T#1m)
	#18 R bOverrideON <= #17.Q
	#19 TOverrideOFF:TON(IN: bOverrideOFF, PT: T#1m)
	#20 R bOverrideOFF <= #19.Q
END_MACRO
#21 MACRO Pump_Sequence(pin 1 "In-1": bPumpSequence)
	#22 AND(NOT LSH405.Q, pin 1)
	#23 AND(LSH405.Q, pin 1)
	#24 AND(#23, NOT #30.ENO, NOT #50.ENO)
	#25 Activate(EN: #24)
	#26 bJokeyPump <= #25
	#27 OR(#22, #29.Q, #34)
	#28 RangeBlock(EN: #23, IN: rWaterPressureSensor, LOWER: 0, UPPER: 3.5)
	#29 Lower_3_5_timer:TON(IN: #28, PT: T#10s)
	#30 Deactivate(EN: #27)
	#31 bJokeyPump <= #30
	#32 bLeadPumpAB <= #30
	#33 bLeadPumpCD <= #30
	#34 AND(#23, PSL412)
	#35 RangeBlock(EN: #23, IN: rWaterPressureSensor, LOWER: 4.7, UPPER: 5.9)
	#36 Activate(EN: #35)
	#37 bLeadPumpAB <= #36
	#38 bLeadPumpCD <= #36
	#39 RangeBlock(EN: #23, IN: rWaterPressureSensor, LOWER: 5.9, UPPER: 6.4)
	#40 Activate(EN: #39)
	#41 bLeadPumpAB <= #40
	#42 bLeadPumpCD <= #43
	#43 Deactivate(EN: #39)
	#44 RangeBlock(EN: #23, IN: rWaterPressureSensor, LOWER: 6.4, UPPER: 8.0)
	#45 Deactivate(EN: #44)
	#46 bLeadPumpAB <= #45
	#47 bLeadPumpCD <= #45
	#48 bJokeyPump <= #50
	#49 RangeBlock(EN: #23, IN: rWaterPressureSensor, LOWER: 8.0, UPPER: 100)
	#50 Deactivate(EN: #49)
	#51 bLeadPumpAB <= #50
	#52 bLeadPumpCD <= #50
	#53 RangeBlock(EN: #23, IN: rWaterPressureSensor, LOWER: 8.2, UPPER: 100)
	#54 Activate(EN: #53)
	#55 bWarningWaterPressureHigh <= #54
END_MACRO
_END_CFC_
(* the same logic as Structured Text *)
input();
(* macro MAINSEQ *)
bVacumPrimingOperation := LSL308A.Q AND LSH308A.Q;
bPumpSequence := LSL308A.Q AND LSH308A.Q;
(* macro VACUM_PRIMING_OPERATION *)
_t1 := (bOverrideON AND bVacumPrimingOperation) OR _t23;
_t4 := _t1 AND NOT _t10 AND NOT bOverrideOFF;
bSolenoidValve := _t4;
bVacumPumDuty := _t4;
_t23 := bVacumPrimingOperation AND NOT LSH405.Q;
WaitToFill(IN := _t1, PT := T#30s);
_t10 := WaitToFill.Q AND NOT FSL101.Q;
bWarning_PrimingNoWater := _t10;
IF bTriggerNegativePressure THEN bOverrideON := TRUE; END_IF;
IF bTriggerPositivePressure THEN bOverrideOFF := TRUE; END_IF;
TOverrideON(IN := bOverrideON, PT := T#1m);
IF TOverrideON.Q THEN bOverrideON := FALSE; END_IF;
TOverrideOFF(IN := bOverrideOFF, PT := T#1m);
IF TOverrideOFF.Q THEN bOverrideOFF := FALSE; END_IF;
(* macro Pump_Sequence *)
_t109 := NOT LSH405.Q AND bPumpSequence;
_t44 := LSH405.Q AND bPumpSequence;
IF _t44 AND NOT _en56 AND NOT _en89 THEN bJokeyPump := Activate(); END_IF;
_t101 := _t109 OR Lower_3_5_timer.Q OR _t102;
IF _t44 THEN _t49 := RangeBlock(IN := rWaterPressureSensor, LOWER := 0, UPPER := 3.5); END_IF;
Lower_3_5_timer(IN := _t49, PT := T#10s);
_en56 := _t101;
IF _en56 THEN _t56 := Deactivate(); END_IF;
IF _en56 THEN bJokeyPump := _t56; END_IF;
IF _en56 THEN bLeadPumpAB := _t56; END_IF;
IF _en56 THEN bLeadPumpCD := _t56; END_IF;
_t102 := _t44 AND PSL412;
IF _t44 THEN _t62 := RangeBlock(IN := rWaterPressureSensor, LOWER := 4.7, UPPER := 5.9); END_IF;
_en65 := _t62;
IF _en65 THEN _t65 := Activate(); END_IF;
IF _en65 THEN bLeadPumpAB := _t65; END_IF;
IF _en65 THEN bLeadPumpCD := _t65; END_IF;
IF _t44 THEN _t68 := RangeBlock(IN := rWaterPressureSensor, LOWER := 5.9, UPPER := 6.4); END_IF;
IF _t68 THEN bLeadPumpAB := Activate(); END_IF;
bLeadPumpCD := _t73;
IF _t68 THEN _t73 := Deactivate(); END_IF;
IF _t44 THEN _t77 := RangeBlock(IN := rWaterPressureSensor, LOWER := 6.4, UPPER := 8.0); END_IF;
_en78 := _t77;
IF _en78 THEN _t78 := Deactivate(); END_IF;
IF _en78 THEN bLeadPumpAB := _t78; END_IF;
IF _en78 THEN bLeadPumpCD := _t78; END_IF;
bJokeyPump := _t89;
IF _t44 THEN _t88 := RangeBlock(IN := rWaterPressureSensor, LOWER := 8.0, UPPER := 100); END_IF;
_en89 := _t88;
IF _en89 THEN _t89 := Deactivate(); END_IF;
bLeadPumpAB := _t89;
bLeadPumpCD := _t89;
IF _t44 THEN _t97 := RangeBlock(IN := rWaterPressureSensor, LOWER := 8.2, UPPER := 100); END_IF;
IF _t97 THEN bWarningWaterPressureHigh := Activate(); END_IF;
END_PROGRAM
ACTION input:
LSH405();
LSL308A();
LSH308A();
FSL101();

rWaterPressureSensor := INT_TO_REAL(PSL411)*(10.0/32767.0);


SolenoidValve_XV102_in := bSolenoidValve;
SolenoidValve_XV102_command := SolenoidValve_XV102_in;
SolenoidValve_XV102_open_Filter(IN:=(NOT SolenoidValve_XV102_status AND SolenoidValve_XV102_in),PT:=T#10s, Q=>SolenoidValve_XV102_open_error);
SolenoidValve_XV102_close_Filter(IN:=( SolenoidValve_XV102_status AND NOT SolenoidValve_XV102_in),PT:=T#10s, Q=>SolenoidValve_XV102_close_error);

SolenoidValve_XV102_common_error := SolenoidValve_XV102_open_error OR SolenoidValve_XV102_close_error;



VacummPump_P403_A_overload_Filter(IN:=(VacummPump_P403_A_overload AND VacummPump_P403_A_in),PT:=T#2s,Q=>VacummPump_P403_A_overload_error);
VacummPump_P403_A_incomplete_Filter(IN:=(VacummPump_P403_A_incomplete AND VacummPump_P403_A_in),PT:=T#2s,Q=>VacummPump_P403_A_incomplete_error);
VacummPump_P403_A_status_Filter(IN:=(NOT VacummPump_P403_A_status AND VacummPump_P403_A_in),PT:=T#10s, Q=>VacummPump_P403_A_status_error);
VacummPump_P403_A_stop_Filter(IN:=( VacummPump_P403_A_status AND NOT VacummPump_P403_A_in),PT:=T#10s, Q=>VacummPump_P403_A_stop_error);

VacummPump_P403_A_common_error := VacummPump_P403_A_overload_error OR VacummPump_P403_A_incomplete_error OR VacummPump_P403_A_status_error OR VacummPump_P403_A_stop_error;


VacummPump_P403_B_overload_Filter(IN:=(VacummPump_P403_B_overload AND VacummPump_P403_B_in),PT:=T#2s,Q=>VacummPump_P403_B_overload_error);
VacummPump_P403_B_incomplete_Filter(IN:=(VacummPump_P403_B_incomplete AND VacummPump_P403_B_in),PT:=T#2s,Q=>VacummPump_P403_B_incomplete_error);
VacummPump_P403_B_status_Filter(IN:=(NOT VacummPump_P403_B_status AND VacummPump_P403_B_in),PT:=T#10s, Q=>VacummPump_P403_B_status_error);
VacummPump_P403_B_stop_Filter(IN:=( VacummPump_P403_B_status AND NOT VacummPump_P403_B_in),PT:=T#10s, Q=>VacummPump_P403_B_stop_error);

VacummPump_P403_B_common_error := VacummPump_P403_B_overload_error OR VacummPump_P403_B_incomplete_error OR VacummPump_P403_B_status_error OR VacummPump_P403_B_stop_error;


VacummPump_P403_A_in := bVacumPumDuty;

VacummPump_P403(
	ERROR1:=VacummPump_P403_A_common_error ,
	ERROR2:=VacummPump_P403_B_common_error ,
	remote1:=VacummPump_P403_A_remote_mode ,
	remote2:=VacummPump_P403_B_remote_mode ,
	IN1:=VacummPump_P403_A_in ,
	IN2:=VacummPump_P403_B_in ,
	Command1=>VacummPump_P403_A_command ,
	Command2=>VacummPump_P403_B_command );

JockeyPump_P402_A_overload_Filter(IN:=(JockeyPump_P402_A_overload AND JockeyPump_P402_A_in),PT:=T#2s,Q=>JockeyPump_P402_A_overload_error);
JockeyPump_P402_A_incomplete_Filter(IN:=(JockeyPump_P402_A_incomplete AND JockeyPump_P402_A_in),PT:=T#2s,Q=>JockeyPump_P402_A_incomplete_error);
JockeyPump_P402_A_status_Filter(IN:=(NOT JockeyPump_P402_A_status AND JockeyPump_P402_A_in),PT:=T#10s, Q=>JockeyPump_P402_A_status_error);
JockeyPump_P402_A_stop_Filter(IN:=( JockeyPump_P402_A_status AND NOT JockeyPump_P402_A_in),PT:=T#10s, Q=>JockeyPump_P402_A_stop_error);

JockeyPump_P402_A_common_error := JockeyPump_P402_A_overload_error OR JockeyPump_P402_A_incomplete_error OR JockeyPump_P402_A_status_error OR JockeyPump_P402_A_stop_error;


JockeyPump_P402_B_overload_Filter(IN:=(JockeyPump_P402_B_overload AND JockeyPump_P402_B_in),PT:=T#2s,Q=>JockeyPump_P402_B_overload_error);
JockeyPump_P402_B_incomplete_Filter(IN:=(JockeyPump_P402_B_incomplete AND JockeyPump_P402_B_in),PT:=T#2s,Q=>JockeyPump_P402_B_incomplete_error);
JockeyPump_P402_B_status_Filter(IN:=(NOT JockeyPump_P402_B_status AND JockeyPump_P402_B_in),PT:=T#10s, Q=>JockeyPump_P402_B_status_error);
JockeyPump_P402_B_stop_Filter(IN:=( JockeyPump_P402_B_status AND NOT JockeyPump_P402_B_in),PT:=T#10s, Q=>JockeyPump_P402_B_stop_error);

JockeyPump_P402_B_common_error := JockeyPump_P402_B_overload_error OR JockeyPump_P402_B_incomplete_error OR JockeyPump_P402_B_status_error OR JockeyPump_P402_B_stop_error;

JockeyPump_P402_A_in := bJokeyPump;

JockeyPump_P402(
	ERROR1:=JockeyPump_P402_A_common_error ,
	ERROR2:=JockeyPump_P402_B_common_error ,
	remote1:=JockeyPump_P402_A_remote_mode ,
	remote2:=JockeyPump_P402_B_remote_mode ,
	IN1:=JockeyPump_P402_A_in ,
	IN2:=JockeyPump_P402_B_in ,
	Command1=>JockeyPump_P402_A_command ,
	Command2=>JockeyPump_P402_B_command );



LeadPump_P401_A_overload_Filter(IN:=(LeadPump_P401_A_overload AND LeadPump_P401_A_in),PT:=T#2s,Q=>LeadPump_P401_A_overload_error);
LeadPump_P401_A_incomplete_Filter(IN:=(LeadPump_P401_A_incomplete AND LeadPump_P401_A_in),PT:=T#2s,Q=>LeadPump_P401_A_incomplete_error);
LeadPump_P401_A_status_Filter(IN:=(NOT LeadPump_P401_A_status AND LeadPump_P401_A_in),PT:=T#10s, Q=>LeadPump_P401_A_status_error);
LeadPump_P401_A_stop_Filter(IN:=( LeadPump_P401_A_status AND NOT LeadPump_P401_A_in),PT:=T#10s, Q=>LeadPump_P401_A_stop_error);

LeadPump_P401_A_common_error := LeadPump_P401_A_overload_error OR LeadPump_P401_A_incomplete_error OR LeadPump_P401_A_status_error OR LeadPump_P401_A_stop_error;


LeadPump_P401_B_overload_Filter(IN:=(LeadPump_P401_B_overload AND LeadPump_P401_B_in),PT:=T#2s,Q=>LeadPump_P401_B_overload_error);
LeadPump_P401_B_incomplete_Filter(IN:=(LeadPump_P401_B_incomplete AND LeadPump_P401_B_in),PT:=T#2s,Q=>LeadPump_P401_B_incomplete_error);
LeadPump_P401_B_status_Filter(IN:=(NOT LeadPump_P401_B_status AND LeadPump_P401_B_in),PT:=T#10s, Q=>LeadPump_P401_B_status_error);
LeadPump_P401_B_stop_Filter(IN:=( LeadPump_P401_B_status AND NOT LeadPump_P401_B_in),PT:=T#10s, Q=>LeadPump_P401_B_stop_error);

LeadPump_P401_B_common_error := LeadPump_P401_B_overload_error OR LeadPump_P401_B_incomplete_error OR LeadPump_P401_B_status_error OR LeadPump_P401_B_stop_error;


LeadPump_P401_C_overload_Filter(IN:=(LeadPump_P401_C_overload AND LeadPump_P401_C_in),PT:=T#2s,Q=>LeadPump_P401_C_overload_error);
LeadPump_P401_C_incomplete_Filter(IN:=(LeadPump_P401_C_incomplete AND LeadPump_P401_C_in),PT:=T#2s,Q=>LeadPump_P401_C_incomplete_error);
LeadPump_P401_C_status_Filter(IN:=(NOT LeadPump_P401_C_status AND LeadPump_P401_C_in),PT:=T#10s, Q=>LeadPump_P401_C_status_error);
LeadPump_P401_C_stop_Filter(IN:=( LeadPump_P401_C_status AND NOT LeadPump_P401_C_in),PT:=T#10s, Q=>LeadPump_P401_C_stop_error);

LeadPump_P401_C_common_error := LeadPump_P401_C_overload_error OR LeadPump_P401_C_incomplete_error OR LeadPump_P401_C_status_error OR LeadPump_P401_C_stop_error;



LeadPump_P401_D_overload_Filter(IN:=(LeadPump_P401_D_overload AND LeadPump_P401_D_in),PT:=T#2s,Q=>LeadPump_P401_D_overload_error);
LeadPump_P401_D_incomplete_Filter(IN:=(LeadPump_P401_D_incomplete AND LeadPump_P401_D_in),PT:=T#2s,Q=>LeadPump_P401_D_incomplete_error);
LeadPump_P401_D_status_Filter(IN:=(NOT LeadPump_P401_D_status AND LeadPump_P401_D_in),PT:=T#10s, Q=>LeadPump_P401_D_status_error);
LeadPump_P401_D_stop_Filter(IN:=( LeadPump_P401_D_status AND NOT LeadPump_P401_D_in),PT:=T#10s, Q=>LeadPump_P401_D_stop_error);

LeadPump_P401_D_common_error := LeadPump_P401_D_overload_error OR LeadPump_P401_D_incomplete_error OR LeadPump_P401_D_status_error OR LeadPump_P401_D_stop_error;

LeadPump_P401_A_in := bLeadPumpAB;
LeadPump_P401_B_in := bLeadPumpAB;

LeadPump_P401_C_in := bLeadPumpCD;
LeadPump_P401_D_in := bLeadPumpCD;

LeadPump_P401_A(
	ERROR1:=LeadPump_P401_A_common_error ,
	remote1:=LeadPump_P401_A_remote_mode ,
	IN1:=LeadPump_P401_A_in ,
	Command1=>LeadPump_P401_A_command );


LeadPump_P401_B(
	ERROR1:=LeadPump_P401_B_common_error ,
	remote1:=LeadPump_P401_B_remote_mode ,
	IN1:=LeadPump_P401_B_in ,
	Command1=>LeadPump_P401_B_command );


LeadPump_P401_C(
	ERROR1:=LeadPump_P401_C_common_error ,
	remote1:=LeadPump_P401_C_remote_mode ,
	IN1:=LeadPump_P401_C_in ,
	Command1=>LeadPump_P401_C_command );


LeadPump_P401_D(
	ERROR1:=LeadPump_P401_D_common_error ,
	remote1:=LeadPump_P401_D_remote_mode ,
	IN1:=LeadPump_P401_D_in ,
	Command1=>LeadPump_P401_D_command );
END_ACTION

(* POU module/Activate, ST *)
FUNCTION Activate : BOOL
VAR_INPUT
END_VAR
VAR
END_VAR
Activate := TRUE;
END_FUNCTION

(* POU module/Deactivate, ST *)
FUNCTION Deactivate : BOOL
VAR_INPUT
END_VAR
VAR
END_VAR
Deactivate := FALSE;
END_FUNCTION

(* POU module/GRIT_REMOVAL_OPERATION_old, CFC *)
PROGRAM GRIT_REMOVAL_OPERATION_old
VAR
	bGritAirBlower: BOOL;
	bGritClasifier: BOOL;
	bSuctionValveOperation: BOOL;
	offGritClassifier: TON;
	B101A: fb_equipment_with_linking;
	bSuctionValveA1: BOOL;
	bSuctionValveA2: BOOL;
	bSuctionValveB1: BOOL;
	bSuctionValveB2: BOOL;
	XV100A: fb_equipment_with_linking;
	XV100B: fb_equipment_with_linking;
	bGritClassifierA: BOOL;
	bGritClassifierB: BOOL;
	C103AandB: fb_equipment_with_linking;
END_VAR
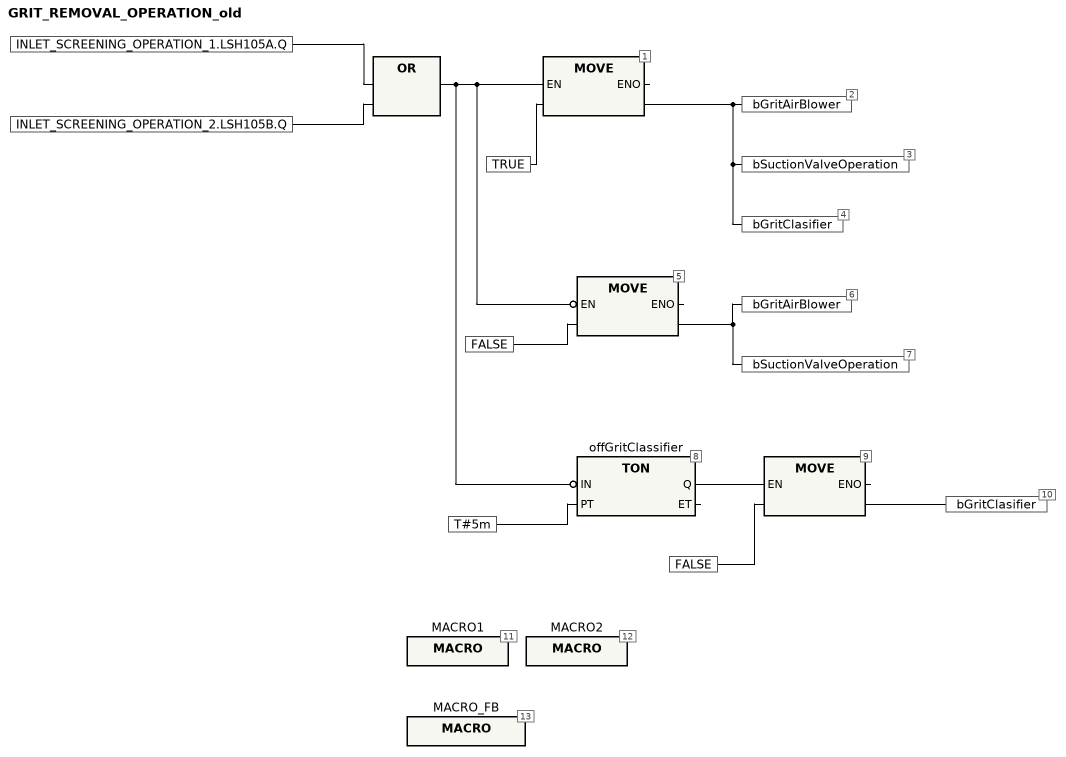
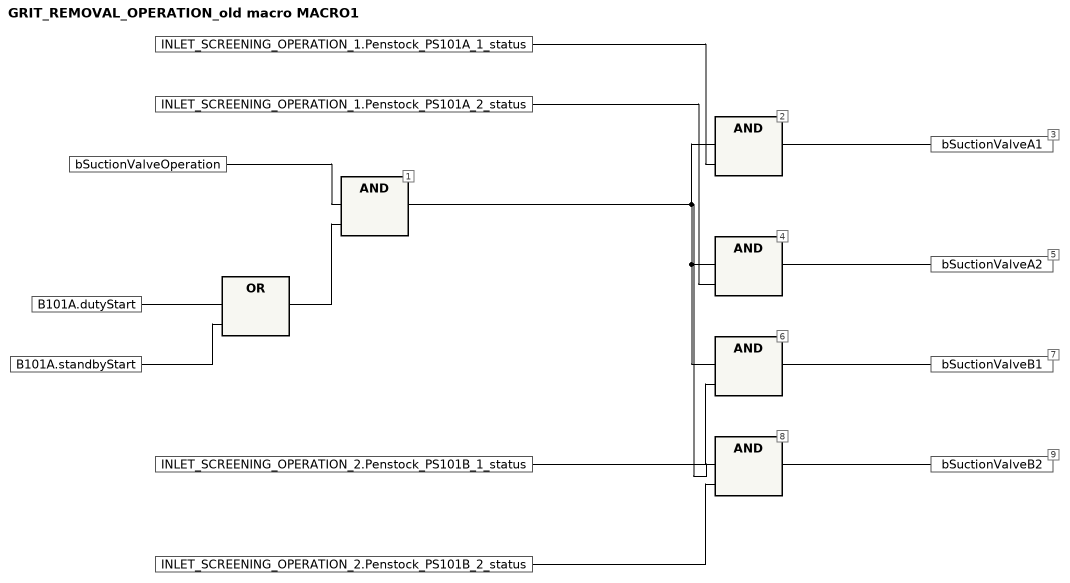
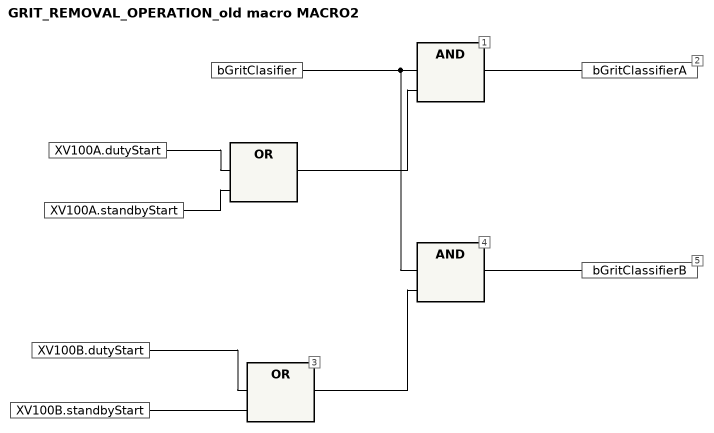
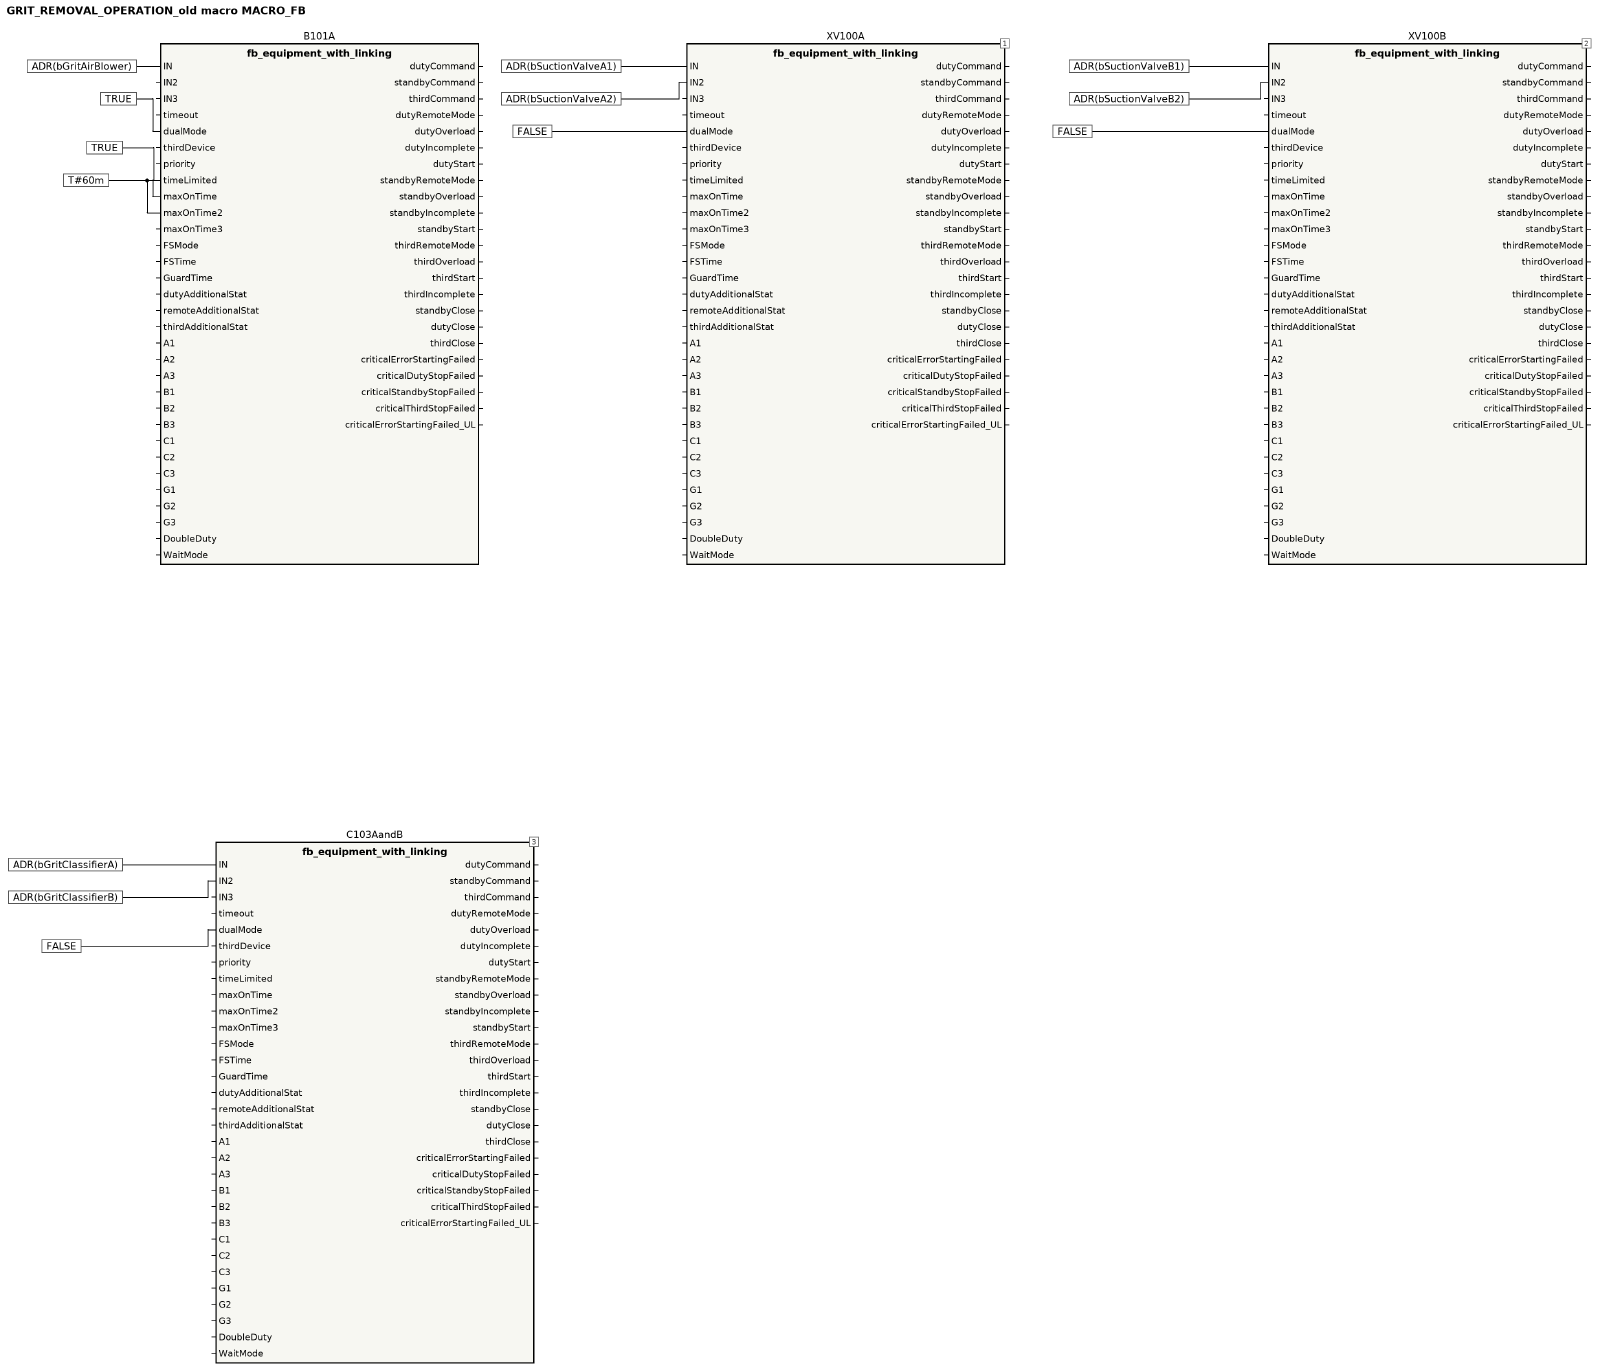
_CFC_ (* Continuous Function Chart, elements in execution order *)
#0 OR(INLET_SCREENING_OPERATION_1.LSH105A.Q, INLET_SCREENING_OPERATION_2.LSH105B.Q)
#1 MOVE(EN: #0, TRUE)
#2 bGritAirBlower <= #1
#3 bSuctionValveOperation <= #1
#4 bGritClasifier <= #1
#5 MOVE(EN: NOT #0, FALSE)
#6 bGritAirBlower <= #5
#7 bSuctionValveOperation <= #5
#8 offGritClassifier:TON(IN: NOT #0, PT: T#5m)
#9 MOVE(EN: #8.Q, FALSE)
#10 bGritClasifier <= #9
#11 MACRO MACRO1()
	#12 OR(B101A.dutyStart, B101A.standbyStart)
	#13 AND(bSuctionValveOperation, #12)
	#14 AND(#13, INLET_SCREENING_OPERATION_1.Penstock_PS101A_1_status)
	#15 bSuctionValveA1 <= #14
	#16 AND(#13, INLET_SCREENING_OPERATION_1.Penstock_PS101A_2_status)
	#17 bSuctionValveA2 <= #16
	#18 AND(#13, INLET_SCREENING_OPERATION_2.Penstock_PS101B_1_status)
	#19 bSuctionValveB1 <= #18
	#20 AND(#13, INLET_SCREENING_OPERATION_2.Penstock_PS101B_2_status)
	#21 bSuctionValveB2 <= #20
END_MACRO
#22 MACRO MACRO2()
	#23 OR(XV100A.dutyStart, XV100A.standbyStart)
	#24 AND(bGritClasifier, #23)
	#25 bGritClassifierA <= #24
	#26 OR(XV100B.dutyStart, XV100B.standbyStart)
	#27 AND(bGritClasifier, #26)
	#28 bGritClassifierB <= #27
END_MACRO
#29 MACRO MACRO_FB()
	#30 B101A:fb_equipment_with_linking(IN: ADR(bGritAirBlower), IN2: -, IN3: -, timeout: -, dualMode: TRUE, thirdDevice: -, priority: -, timeLimited: TRUE, maxOnTime: T#60m, maxOnTime2: T#60m, maxOnTime3: -, FSMode: -, FSTime: -, GuardTime: -, dutyAdditionalStat: -, remoteAdditionalStat: -, thirdAdditionalStat: -, A1: -, A2: -, A3: -, B1: -, B2: -, B3: -, C1: -, C2: -, C3: -, G1: -, G2: -, G3: -, DoubleDuty: -, WaitMode: -)
	#31 XV100A:fb_equipment_with_linking(IN: ADR(bSuctionValveA1), IN2: ADR(bSuctionValveA2), IN3: -, timeout: -, dualMode: FALSE, thirdDevice: -, priority: -, timeLimited: -, maxOnTime: -, maxOnTime2: -, maxOnTime3: -, FSMode: -, FSTime: -, GuardTime: -, dutyAdditionalStat: -, remoteAdditionalStat: -, thirdAdditionalStat: -, A1: -, A2: -, A3: -, B1: -, B2: -, B3: -, C1: -, C2: -, C3: -, G1: -, G2: -, G3: -, DoubleDuty: -, WaitMode: -)
	#32 XV100B:fb_equipment_with_linking(IN: ADR(bSuctionValveB1), IN2: ADR(bSuctionValveB2), IN3: -, timeout: -, dualMode: FALSE, thirdDevice: -, priority: -, timeLimited: -, maxOnTime: -, maxOnTime2: -, maxOnTime3: -, FSMode: -, FSTime: -, GuardTime: -, dutyAdditionalStat: -, remoteAdditionalStat: -, thirdAdditionalStat: -, A1: -, A2: -, A3: -, B1: -, B2: -, B3: -, C1: -, C2: -, C3: -, G1: -, G2: -, G3: -, DoubleDuty: -, WaitMode: -)
	#33 C103AandB:fb_equipment_with_linking(IN: ADR(bGritClassifierA), IN2: ADR(bGritClassifierB), IN3: -, timeout: -, dualMode: FALSE, thirdDevice: -, priority: -, timeLimited: -, maxOnTime: -, maxOnTime2: -, maxOnTime3: -, FSMode: -, FSTime: -, GuardTime: -, dutyAdditionalStat: -, remoteAdditionalStat: -, thirdAdditionalStat: -, A1: -, A2: -, A3: -, B1: -, B2: -, B3: -, C1: -, C2: -, C3: -, G1: -, G2: -, G3: -, DoubleDuty: -, WaitMode: -)
END_MACRO
_END_CFC_
END_PROGRAM

(* POU module/fb_equipment_with_linking, ST *)
FUNCTION_BLOCK fb_equipment_with_linking
VAR_INPUT
	IN							: POINTER TO BOOL;
	IN2							: POINTER TO BOOL;
	IN3							: POINTER TO BOOL;

	timeout						: TIME:= T#2s;
	dualMode					: BOOL:=TRUE;
	thirdDevice					: BOOL:= FALSE;
	priority						: BOOL := FALSE;
	timeLimited					: BOOL :=FALSE;
	maxOnTime					: TIME := T#10s;
	maxOnTime2					: TIME := T#10s;
	maxOnTime3					: TIME := T#10s;

	FSMode						: BOOL := FALSE;
	FSTime						: TIME := T#2m;
(*
	FSBothTime					: TIME := T#5m;
*)
	GuardTime					: TIME := T#5m;




	dutyAdditionalStat				AT%I* : BOOL := TRUE;
	remoteAdditionalStat			AT%I* : BOOL := TRUE;
	thirdAdditionalStat				AT%I* : BOOL := TRUE;

	A1							: POINTER TO BOOL;
	A2							: POINTER TO BOOL;
	A3							: POINTER TO BOOL;
	B1							: POINTER TO BOOL;
	B2							: POINTER TO BOOL;
	B3							: POINTER TO BOOL;
	C1							: POINTER TO BOOL;
	C2							: POINTER TO BOOL;
	C3							: POINTER TO BOOL;
(*
	Q1							: POINTER TO BOOL;
	Q2							: POINTER TO BOOL;
	Q3							: POINTER TO BOOL;
*)
	G1							: POINTER TO BOOL;
	G2							: POINTER TO BOOL;
	G3							: POINTER TO BOOL;

	DoubleDuty: BOOL;
	WaitMode : BOOL;
END_VAR
VAR_OUTPUT

	dutyCommand				AT%Q*: BOOL;
	standbyCommand				AT%Q*: BOOL;
	thirdCommand				AT%Q*: BOOL;

	dutyRemoteMode				AT%I* : BOOL;
	dutyOverload					AT%I* : BOOL;
	dutyIncomplete				AT%I* : BOOL;
	dutyStart						AT%I* : BOOL;

	standbyRemoteMode			AT%I* : BOOL;
	standbyOverload				AT%I* : BOOL;
	standbyIncomplete			AT%I* : BOOL;
	standbyStart					AT%I* : BOOL;

	thirdRemoteMode				AT%I* : BOOL;
	thirdOverload					AT%I* : BOOL;
	thirdStart						AT%I* : BOOL;
	thirdIncomplete				AT%I* : BOOL;

	standbyClose					AT%I* : BOOL;
	dutyClose					AT%I* : BOOL;
	thirdClose					AT%I* : BOOL;


	criticalErrorStartingFailed		: BOOL;
	criticalDutyStopFailed			: BOOL;
	criticalStandbyStopFailed		: BOOL;
	criticalThirdStopFailed			: BOOL;

	criticalErrorStartingFailed_UL	: BOOL;


END_VAR
VAR




	warningDutyOverload			: BOOL;
	warningDutyFailed				: BOOL;
	warningDutyNotClose			: BOOL;
	warningDutyClose				: BOOL;
	warningStandbyOverload		: BOOL;
	warningStandbyFailed			: BOOL;
	warningStandbyNotClose		: BOOL;
	warningStandbyClose			: BOOL;
	warningThirdOverload			: BOOL;
	warningThirdFailed			: BOOL;
	warningThirdNotClose			: BOOL;
	warningThirdClose			: BOOL;

	duty							: INT;
	iStopDuty					: INT;
	state						: INT;
	third							: INT;
	iStopThird					: INT;
	iStopStandby					: INT;
	standby						: INT;
	startDuty						: BOOL;
	startStandby					: BOOL;
	stopStandby					: BOOL;
	stopDuty						: BOOL;
	dutyHalt						: BOOL;
	standbyHalt					: BOOL;
	stopThird					: BOOL;
	startThird					: BOOL;
	thirdHalt						: BOOL;

	dutyTimer					: TON;
	standbyTimer					: TON;
	stopStandbyTimer				: TON;
	stopDutyTimer				: TON;
	FSStopDuty					:TON;
	FSStopStandby				: TON;
	FSBothStop					: TON;
	OnTimer						: TON;
	StandbyOnTimer				: TON;
	thirdTimer					: TON;
	stopThirdTimer				: TON;
	GuardTONDuty				: TON;
	GuardTONStandby			: TON;
	GuardTONThird				: TON;

	ROnce5						: R_TRIG;
	ROnce10					: R_TRIG;
	ROnce20					: R_TRIG;
	SOnceDuty					: R_TRIG;
	SOnceStandby				: R_TRIG;
	SOnceFS					: R_TRIG;
	SOnceThird					: R_TRIG;
	DutyStopR					: R_TRIG;
	StandbyStopR				: R_TRIG;
	ThirdStopR					: R_TRIG;

	internalDummy: BOOL;
	dummyIN: BOOL;
	dummyIN2: BOOL;
	dummyIN3: BOOL;
END_VAR
VAR_IN_OUT
END_VAR
IF WaitMode THEN
	standbyRemoteMode			:=TRUE;
	standbyStart					:=TRUE;

	thirdRemoteMode				:=TRUE;

	thirdIncomplete				:=TRUE;
END_IF

IF IN = 0 THEN
	IN := ADR(dummyIN);
END_IF

IF IN2 = 0 THEN
	IN2 := ADR(dummyIN2);
END_IF

IF IN3 = 0 THEN
	IN3 := ADR(dummyIN3);
END_IF

IF A1 = 0 THEN
	A1 := ADR(internalDummy);
END_IF
IF A2 = 0 THEN
	A2 := ADR(internalDummy);
END_IF
IF A3 = 0 THEN
	A3 := ADR(internalDummy);
END_IF

IF B1 = 0 THEN
	B1 := ADR(internalDummy);
END_IF
IF B2 = 0 THEN
	B2 := ADR(internalDummy);
END_IF
IF B3 = 0 THEN
	B3 := ADR(internalDummy);
END_IF

IF C1 = 0 THEN
	C1 := ADR(internalDummy);
END_IF
IF C2 = 0 THEN
	C2 := ADR(internalDummy);
END_IF
IF C3 = 0 THEN
	C3 := ADR(internalDummy);
END_IF

IF G1 = 0 THEN
	G1 := ADR(internalDummy);
END_IF
IF G2 = 0 THEN
	G2 := ADR(internalDummy);
END_IF
IF G3 = 0 THEN
	G3 := ADR(internalDummy);
END_IF


(*
IF warningDutyOverload = 0 THEN
	warningDutyOverload := ADR(internalDummy);
END_IF
IF warningDutyFailed = 0 THEN
	warningDutyFailed := ADR(internalDummy);
END_IF
IF warningDutyNotClose = 0 THEN
	warningDutyNotClose := ADR(internalDummy);
END_IF
IF warningDutyClose = 0 THEN
	warningDutyClose := ADR(internalDummy);
END_IF



IF warningStandbyOverload = 0 THEN
	warningStandbyOverload := ADR(internalDummy);
END_IF
IF warningStandbyFailed = 0 THEN
	warningStandbyFailed := ADR(internalDummy);
END_IF
IF warningStandbyNotClose = 0 THEN
	warningStandbyNotClose := ADR(internalDummy);
END_IF
IF warningStandbyClose = 0 THEN
	warningStandbyClose := ADR(internalDummy);
END_IF


IF warningThirdOverload = 0 THEN
	warningThirdOverload := ADR(internalDummy);
END_IF
IF warningThirdFailed = 0 THEN
	warningThirdFailed := ADR(internalDummy);
END_IF
IF warningThirdNotClose = 0 THEN
	warningThirdNotClose := ADR(internalDummy);
END_IF
IF warningThirdClose = 0 THEN
	warningThirdClose := ADR(internalDummy);
END_IF


IF criticalErrorStartingFailed = 0 THEN
	criticalErrorStartingFailed := ADR(internalDummy);
END_IF
IF criticalDutyStopFailed = 0 THEN
	criticalDutyStopFailed := ADR(internalDummy);
END_IF
IF criticalStandbyStopFailed = 0 THEN
	criticalStandbyStopFailed := ADR(internalDummy);
END_IF
IF criticalThirdStopFailed = 0 THEN
	criticalThirdStopFailed := ADR(internalDummy);
END_IF
*)
(*---------------------------------------------------------------------------------------------------------------------------*)

IF dualMode THEN

IF NOT IN^ THEN
	state := 0;
	stopDuty := TRUE;
	stopStandby := TRUE;

	startDuty:=FALSE;
	startStandby := FALSE;
	IF thirdDevice THEN
		stopThird :=TRUE;
		startThird := FALSE;
	END_IF
END_IF

ELSE

state := 0;
startDuty := IN^;
stopDuty := NOT IN^;

startStandby := IN2^;
stopStandby := NOT IN2^;

startThird := IN3^;
stopThird := NOT IN3^;

A1^:=  IN^;
A2^:= IN^;
A3^ := IN^;
B1^:=  IN2^;
B2^:= IN2^;
B3^ := IN2^;
C1^:=  IN3^;
C2^:= IN3^;
C3^ := IN3^;

END_IF

(*
IF NOT IN^ THEN
	state := 0;
	stopDuty := TRUE;
	stopStandby := TRUE;

	startDuty:=FALSE;
	startStandby := FALSE;
	IF thirdDevice THEN
		stopThird :=TRUE;
		startThird := FALSE;
	END_IF
ELSIF IN^ AND NOT dualMode THEN
	state := 0;
	stopDuty := FALSE;
	stopStandby := FALSE;

	startDuty:=TRUE;
	startStandby := TRUE;
	IF thirdDevice THEN
		stopThird :=FALSE;
		startThird := TRUE;
	END_IF

	A1^:= TRUE;
	A2^:=TRUE;
	A3^ :=TRUE;
	B1^:= TRUE;
	B2^:=TRUE;
	B3^ :=TRUE;
	C1^:= TRUE;
	C2^:=TRUE;
	C3^ :=TRUE;
END_IF
*)

(*-------------------------------------------------------------------------------------------------------------------------------------------*)

IF NOT DoubleDuty THEN

CASE state OF
0:
	state := 5;
5:
	IF NOT DutyHalt AND dutyStart THEN
		stopStandby := TRUE;
		stopThird:=TRUE;
	END_IF

	stopDuty := FALSE;
	startDuty := TRUE;
	IF timeLimited THEN
		OnTimer(IN:=TRUE,PT:=maxOnTime);
	ELSE
		OnTimer(IN:=FALSE,PT:=maxOnTime);
	END_IF
	IF dutyHalt  OR onTimer.Q THEN
		OnTimer(IN:=FALSE,PT:=maxOnTime);
		startDuty := FALSE;
		stopDuty := TRUE;
		state := 10;
	END_IF
10:
	IF NOT StandbyHalt AND standbyStart THEN
		stopDuty := TRUE;
		stopThird:=TRUE;
	END_IF

	stopStandby := FALSE;
	startStandby := TRUE;

	IF timeLimited THEN
		OnTimer(IN:=TRUE,PT:=maxOnTime2);
	ELSE
		OnTimer(IN:=FALSE,PT:=maxOnTime2);
	END_IF
	IF standbyHalt OR onTimer.Q THEN
		OnTimer(IN:=FALSE,PT:=maxOnTime2);
		startStandby := FALSE;
		stopStandby := TRUE;
		IF thirdDevice THEN
			IF priority THEN
				IF dutyIncomplete OR dutyOverload THEN
					state:= 20;
				ELSE
					dutyHalt := FALSE;
					standbyHalt := FALSE;
					state:=0;
				END_IF
			ELSE
				state:= 20;
			END_IF
		ELSE
			IF dutyIncomplete OR dutyOverload THEN
				CriticalErrorStartingFailed := TRUE;
			END_IF
			state:=0;
			dutyHalt := FALSE;
			standbyHalt := FALSE;
		END_IF
	END_IF
20:
	IF NOT thirdHalt AND thirdStart THEN
		stopStandby := TRUE;
		stopDuty:=TRUE;
	END_IF

	stopThird := FALSE;
	startThird := TRUE;
	IF timeLimited THEN
		OnTimer(IN:=TRUE,PT:=maxOnTime3);
	ELSE
		OnTimer(IN:=FALSE,PT:=maxOnTime3);
	END_IF
	IF thirdHalt OR OnTimer.Q THEN
		OnTimer(IN:=FALSE,PT:=maxOnTime3);
		startThird := FALSE;
		stopThird := TRUE;
		state := 0;
		IF  (dutyIncomplete OR dutyOverload)  AND (standbyIncomplete OR standbyOverload) THEN
				CriticalErrorStartingFailed := TRUE;
		END_IF
		dutyHalt := FALSE;
		standbyHalt := FALSE;
		thirdHalt := FALSE;
	END_IF
END_CASE

ELSE

thirdDevice := TRUE; (*third device must be enable when double duty*)
dualMode := TRUE; (*dual mode also must be true*)

CASE state OF
0:
	state := 5;
5:
	thirdHalt := FALSE;
	stopStandby := TRUE;
	startStandby := FALSE;

	stopDuty := FALSE;
	startDuty := TRUE;

	stopThird := FALSE;
	startThird := TRUE;

	IF dutyHalt  THEN
		state := 10;
	END_IF


	IF thirdHalt  THEN
		state := 20;
	END_IF
10:
	dutyHalt := FALSE;

	stopStandby := FALSE;
	startStandby := TRUE;

	stopDuty := TRUE;
	startDuty := FALSE;

	stopThird := FALSE;
	startThird := TRUE;

	IF standbyHalt THEN
		state:= 0;
	END_IF
20:
	thirdHalt := FALSE;

	stopStandby := FALSE;
	startStandby := TRUE;

	stopDuty := FALSE;
	startDuty := TRUE;

	stopThird := TRUE;
	startThird := FALSE;

	IF standbyHalt THEN
		state:= 0;
	END_IF
END_CASE


IF NOT(state = 0) AND  (dutyIncomplete OR dutyOverload)  AND (standbyIncomplete OR standbyOverload) AND (thirdIncomplete OR thirdOverload)  THEN
	CriticalErrorStartingFailed := TRUE;
	criticalErrorStartingFailed_UL := TRUE;
ELSE
	criticalErrorStartingFailed_UL := FALSE;
END_IF
END_IF

(*-------------------------------------------------------------------------------------------------------------------------------------------*)

CASE duty OF
0:
	IF startDuty THEN
		duty := 5;
	END_IF
5:
	IF dutyRemoteMode AND dutyAdditionalStat THEN
		duty := 10;
	ELSE
		duty := 900;
	END_IF
10:
	IF dutyOverload THEN
		warningDutyOverload := TRUE;
		dutyHalt := TRUE;
		duty := 40;
	ELSE
		duty := 15;
	END_IF

15:
	duty := 20;
	dutyCommand := TRUE;
20:
	dutyTimer(IN:= TRUE, PT := timeout);
	IF dutyTimer.Q THEN
		dutyTimer(IN:=FALSE);
		duty := 30;
	END_IF
30:

		IF dutyIncomplete OR NOT dutyStart THEN
			warningDutyFailed := TRUE;
			dutyHalt := TRUE;
			IF  dutyClose THEN
				warningDutyClose := TRUE;
			END_IF
		END_IF
		duty := 40;
40:

	duty := 900;
900:
	duty := 0;
END_CASE

(*----------------------------------------------------------------------------------------------------------------------*)

CASE standby OF
0:
	IF startStandby THEN
		standby := 5;
	END_IF
5:
	IF standbyRemoteMode AND remoteAdditionalStat THEN
		standby := 10;
	ELSE
		standby := 900;
	END_IF
10:
	IF standbyOverload THEN
		warningStandbyOverload := TRUE;
		standbyHalt := TRUE;
		standby := 40;
	ELSE
		standby := 15;
	END_IF
15:
		standbyCommand := TRUE;
		standby := 20;
20:
	standbyTimer(IN:= TRUE, PT := timeout);
	IF standbyTimer.Q THEN
		standbyTimer(IN:=FALSE);
		standby := 30;
	END_IF
30:

		IF standbyIncomplete OR NOT standbyStart THEN
			warningStandbyFailed := TRUE;
			standbyHalt := TRUE;
			IF  standbyClose THEN
				warningStandbyClose := TRUE;
			END_IF
		END_IF
		standby := 40;
40:

	standby := 900;

900:
	standby := 0;
END_CASE

(*-------------------------------------------------------------------------------------------------------------------------------------------*)

CASE third OF
0:
	IF startThird THEN
		third := 5;
	END_IF
5:
	IF thirdRemoteMode AND thirdAdditionalStat THEN
		third := 10;
	ELSE
		third := 900;
	END_IF
10:
	IF thirdOverload THEN
		warningThirdOverload := TRUE;
		thirdHalt := TRUE;
		third := 40;
	ELSE
		third := 15;
	END_IF
15:
		thirdCommand := TRUE;
		third := 20;
20:
	thirdTimer(IN:= TRUE, PT := timeout);
	IF thirdTimer.Q THEN
		thirdTimer(IN:=FALSE);
		third := 30;
	END_IF
30:

		IF thirdIncomplete OR NOT thirdStart THEN
			warningThirdFailed := TRUE;
			thirdHalt := TRUE;
			IF thirdClose THEN
				warningThirdClose := TRUE;
			END_IF
		END_IF
		third := 40;
40:

	third := 900;

900:
	third := 0;
END_CASE

(*-------------------------------------------------------------------------------------------------------------------------------------------*)

ROnce5(CLK:=(state=5));
IF ROnce5.Q THEN
		A1^:= TRUE;
		A2^:=TRUE;
		A3^ :=TRUE;
END_IF

ROnce10(CLK:=(state=10));
IF ROnce10.Q THEN
		B1^:= TRUE;
		B2^:= TRUE;
		B3^:= TRUE;
END_IF

IF thirdDevice THEN
ROnce20(CLK:=(state=20));
IF ROnce20.Q THEN
		C1^:= TRUE;
		C2^:= TRUE;
		C3^:= TRUE;
END_IF
END_IF

(*-------------------------------------------------------------------------------------------------------------------------------------------*)
GuardTONDuty(IN:=dutyIncomplete OR dutyOverload OR NOT dutyStart, PT:= GuardTime);
IF GuardTONDuty.Q THEN
	G1^ := TRUE;
END_IF
GuardTONStandby(IN:=standbyIncomplete OR standbyOverload OR NOT standbyStart, PT:= GuardTime);
IF GuardTONStandby.Q THEN
	G2^ := TRUE;
END_IF

IF thirdDevice THEN
GuardTONThird(IN:=thirdIncomplete OR thirdOverload OR NOT thirdStart, PT:= GuardTime);
IF GuardTONThird.q THEN
	G3^ := TRUE;
END_IF
END_IF
(*-------------------------------------------------------------------------------------------------------------------------------------------*)
stopAction;
test();
END_FUNCTION_BLOCK
ACTION stopAction:
CASE iStopDuty OF
0:
	DutyStopR(CLK:=stopDuty);
	IF DutyStopR.Q THEN
		iStopDuty := 5;
	END_IF
5:
	IF FSMode THEN
		FSStopDuty(IN:=TRUE,PT:=FSTime);
		IF FSStopDuty.Q THEN
			iStopDuty := 10;
			FSStopDuty(IN:=FALSE,PT:=FSTime);
		END_IF
	ELSE
		iStopDuty:=10;
	END_IF
10:
	dutyCommand := FALSE;
	stopDutyTimer(IN:=TRUE, PT:=timeout);
		IF stopDutyTimer.Q THEN
			stopDutyTimer(IN:=FALSE);
			IF NOT dutyClose THEN
				IF dutyStart THEN
					criticalDutyStopFailed := TRUE;
				END_IF
				warningDutyNotClose := TRUE;
			END_IF
			iStopDuty := 0;
		END_IF
END_CASE

(*-------------------------------------------------------------------------------------------------------------------------------------------*)

